	bAutomat4 := fbButtAuto4.bOutB  AND NOT bStartAutomat4 AND NOT bSound4;
	fbPuls(tPeriod := T#0.5S);

	fbButtManu4(bButt := bButtManu4 AND NOT  bAutomat4, bReset := bReset4 OR bAlarm4);
	bManual4 := fbButtManu4.bOutB;

	fbButtReverse4(bButt := bButtReverse4 AND NOT b_4KM1_1, bReset := bReset4 OR bAlarm4);
	bReverse4 := fbButtReverse4.bOutB;

	fbButtStop4(bButt := bButtStop4 OR bAlarm4, bReset := bReset4);
	bStop4 := fbButtStop4.bOutB ;
    	
	fbTimerStart4 (IN := bStartAutomat4, PT := T#1S);

IF NOT bStop4 AND fbTimerStart4.Q AND NOT 
  ( bDrive4s01M1 OR bDrive4s02M1 OR bDrive4s03M1 OR 
	bDrive4s04M1 OR bDrive4s05M1 OR bDrive4s06M1 OR 
	bDrive4s01M1Rev OR bDrive4s02M1Rev OR bDrive4s03M1Rev OR 
	bDrive4s04M1Rev OR bDrive4s05M1Rev OR bDrive4s06M1Rev )
THEN bStartAutomat4 := FALSE;
END_IF

IF bReset4 THEN bAutomat4 := FALSE; bManual4 := FALSE; bStop4 := FALSE; bStartAutomat4 := FALSE;
END_IF

fbpulse4(ENABLE := bStartAutomat4 OR bSound4,TIMELOW := T#500MS, TIMEHIGH:=T#500MS);
//Светофоры первого конвейера
bGreen_4S1HL1  := bAutomat4 AND NOT bManual4 AND NOT bAlarm4 AND NOT bSound4 OR fbpulse4.OUT;
bGreen_4S1_HL1 := bAutomat4 AND NOT bManual4 AND NOT bAlarm4 AND NOT bSound4 OR fbpulse4.OUT;

bYellow_4S1HL1 := NOT bAutomat4 AND bManual4 AND NOT bAlarm4;
bYellow_4S1_HL1:= NOT bAutomat4 AND bManual4 AND NOT bAlarm4;
//---------------------------------------------------------------------------------------------------//

ACTION ACT_Conversion:
Massa_1_INT :=REAL_TO_INT( Massa_1);
Massa_2_INT :=REAL_TO_INT( Massa_2);
Massa_3_INT :=REAL_TO_INT( Massa_3);
Massa_4_INT :=REAL_TO_INT( Massa_4);

Massa_1_Gramms := REAL_TO_DINT( Massa_1 * 1000000);
Massa_2_Gramms := REAL_TO_DINT( Massa_2 * 1000000);
Massa_3_Gramms := REAL_TO_DINT( Massa_3 * 1000000);
Massa_4_Gramms := REAL_TO_DINT( Massa_4 * 1000000);
END_ACTION

ACTION ACT_Drive:
//----------------------------------------------------------// конвейер 1
b1K2 := bDrive1s01M1 OR bDrive1s01M1Rev; // Пуск 1UZ1					 
b1K3 := bDrive1s02M1 OR bDrive1s02M1Rev; // Пуск 1UZ2
b1K4 := bDrive1s03M1 OR bDrive1s03M1Rev; // Пуск 1UZ3
b1K5 := bDrive1s04M1 OR bDrive1s04M1Rev; // Пуск 1UZ4
b1K6 := bDrive1s05M1 OR bDrive1s05M1Rev; // Пуск 1UZ5
b1K7 := bDrive1s06M1 OR bDrive1s06M1Rev; // Пуск 1UZ6
//---------------------------------------------------------// конвейер 2
b2K2 := bDrive2s01M1 OR bDrive2s01M1Rev; // Пуск 2UZ1					 
b2K3 := bDrive2s02M1 OR bDrive2s02M1Rev; // Пуск 2UZ2
b2K4 := bDrive2s03M1 OR bDrive2s03M1Rev; // Пуск 2UZ3
b2K5 := bDrive2s04M1 OR bDrive2s04M1Rev; // Пуск 2UZ4
b2K6 := bDrive2s05M1 OR bDrive2s05M1Rev; // Пуск 2UZ5
b2K7 := bDrive2s06M1 OR bDrive2s06M1Rev; // Пуск 2UZ6
//---------------------------------------------------------// конвейер 3
b3K2 := bDrive3s01M1 OR bDrive3s01M1Rev; // Пуск 3UZ1					 
b3K3 := bDrive3s02M1 OR bDrive3s02M1Rev; // Пуск 3UZ2
b3K4 := bDrive3s03M1 OR bDrive3s03M1Rev; // Пуск 3UZ3
b3K5 := bDrive3s04M1 OR bDrive3s04M1Rev; // Пуск 3UZ4
b3K6 := bDrive3s05M1 OR bDrive3s05M1Rev; // Пуск 3UZ5
b3K7 := bDrive3s06M1 OR bDrive3s06M1Rev; // Пуск 3UZ6
//---------------------------------------------------------// конвейер 4
b4K2 := bDrive4s01M1 OR bDrive4s01M1Rev; // Пуск 4UZ1					 
b4K3 := bDrive4s02M1 OR bDrive4s02M1Rev; // Пуск 4UZ2
b4K4 := bDrive4s03M1 OR bDrive4s03M1Rev; // Пуск 4UZ3
b4K5 := bDrive4s04M1 OR bDrive4s04M1Rev; // Пуск 4UZ4
b4K6 := bDrive4s05M1 OR bDrive4s05M1Rev; // Пуск 4UZ5
b4K7 := bDrive4s06M1 OR bDrive4s06M1Rev; // Пуск 4UZ6
END_ACTION

ACTION ACT_Light:
bSound_1S1HL1 := bSound1;
bSound_1S1_HL1:= bSound1;
bSound_2S1HL1 := bSound2;
bSound_2S1_HL1:= bSound2;
bSound_3S1HL1 := bSound3;
bSound_3S1_HL1:= bSound3;
bSound_4S1HL1 :=bSound4;
bSound_4S1_HL1:=bSound4;
END_ACTION

END_PROGRAM

// ---- POUs/FB/Puls.TcPOU
FUNCTION_BLOCK Puls

VAR_INPUT
 	EN 		:BOOL := TRUE;
    Period	:TIME;
END_VAR
VAR_OUTPUT
	Puls	:BOOL;
END_VAR
VAR
	M		:BOOL:=0;
	R1		:R_TRIG;
	t		:BOOL;
	R2		:R_TRIG;
	TP1		:TP;
	TP2		:TP;
	M1		:BOOL:=0;
END_VAR

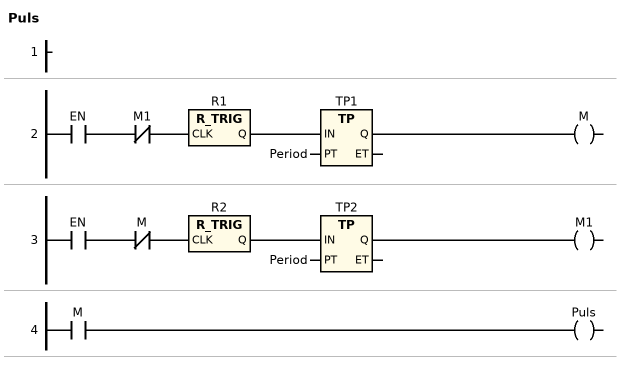
// NETWORK 1

// NETWORK 2
R1(CLK := EN AND NOT M1); // R_TRIG
TP1(IN := R1.Q, PT := Period); // TP
M := TP1.Q;

// NETWORK 3
R2(CLK := EN AND NOT M); // R_TRIG
TP2(IN := R2.Q, PT := Period); // TP
M1 := TP2.Q;

// NETWORK 4
Puls := M;

END_FUNCTION_BLOCK

// ---- POUs/FB/FBauxiliary/FB_ButtonToggle.TcPOU
FUNCTION_BLOCK FB_ButtonToggle
VAR_INPUT
	bReset  :BOOL;
	bEnable :BOOL := TRUE;
	bButt   :BOOL;
END_VAR
VAR
	fbButt  :R_TRIG;
END_VAR
VAR_OUTPUT
	bOutB   :BOOL;
END_VAR

fbButt(CLK:=bButt);

IF fbButt.Q AND bEnable THEN
	IF bOutB THEN bOutB := FALSE;
		ELSE bOutB := TRUE;
	END_IF
END_IF

IF bReset THEN bOutB := FALSE;
END_IF

END_FUNCTION_BLOCK

// ---- POUs/FB/FB_Puls.TcPOU
FUNCTION_BLOCK FB_Puls
VAR_INPUT
	tPeriod  :TIME;
END_VAR
VAR_OUTPUT
	bPuls 	 :BOOL;
END_VAR
VAR
	bM1		 :BOOL := TRUE;
	TP1		 :TP;
	TP2		 :TP;
	fbPulsM1 :F_TRIG;
	iCounter :INT;
	bM2		 :BOOL;
	fbPulsM2 :F_TRIG;
END_VAR

fbPulsM1(CLK:= bM1);
TP1(IN:= fbPulsM1.Q, PT:=tPeriod);
bM2 :=TP1.Q;

fbPulsM2(CLK:= bM2);
TP2(IN:= fbPulsM1.Q,  PT:=tPeriod);

bM1:= TP2.Q;
bPuls := bM1;
IF fbPulsM1.Q THEN
	iCounter:=iCounter+1;
END_IF

END_FUNCTION_BLOCK

// ---- POUs/TCP_IP.TcPOU
PROGRAM TCP_IP
VAR		 
	sSrvNetID	:T_AmsNetID := '';						/// TwinCAT TCP/IP server network address
	sLocalHost	:T_IPv4Addr := '10.45.19.80';			/// Own (server) IP address! 
	 
	nLocalPort1	:UDINT := 2001;							/// Own (server 1) port number!	
	nLocalPort2	:UDINT := 2002;							/// Own (server 2) port number!  
	nLocalPort3	:UDINT := 2003;							/// Own (server 3) port number!	 
	nLocalPort4	:UDINT := 2004;							/// Own (server 4) port number!
	 
	bEnable1	:BOOL  := TRUE;							/// TRUE => enable server 1(connection) instance, FALSE => disable
	bEnable2	:BOOL  := TRUE;							/// TRUE => enable server 2(connection) instance, FALSE => disable
	bEnable3	:BOOL  := TRUE;							/// TRUE => enable server 3(connection) instance, FALSE => disable
	bEnable4	:BOOL  := TRUE;							/// TRUE => enable server 4(connection) instance, FALSE => disable
	bEnable5	:BOOL  := TRUE;							/// TRUE => enable server  (connection) instance, FALSE => disable
	
	bLog		:BOOL  := TRUE;							/// TRUE => Enable error/message log, FALSE => Disable 
	 
	fbServer1	:FB_Server := (sPrefix := 'SERVER1::');	/// Application (connection) instance 1
	fbServer2	:FB_Server := (sPrefix := 'SERVER2::');	/// Application (connection) instance 2
	fbServer3	:FB_Server := (sPrefix := 'SERVER3::');	/// Application (connection) instance 3
	fbServer4	:FB_Server := (sPrefix := 'SERVER4::');	/// Application (connection) instance 4
	 
	hServer1	:T_HSERVER;								/// Server connection handle 1	
	hServer2	:T_HSERVER;								/// Server connection handle 2	
	hServer3	:T_HSERVER;								/// Server connection handle 3
	hServer4	:T_HSERVER; 							/// Server connection handle 4

	fbCloseAll	:FB_SocketCloseAll;
	bInitialize	:BOOL := TRUE;

END_VAR

IF bInitialize THEN
	bInitialize := FALSE;

	(* Initialize server handle once *)
	F_CreateServerHnd( 	sSrvNetID 	:= sSrvNetID, 
						sLocalHost 	:= sLocalHost, 
						nLocalPort	:= nLocalPort1,
						nMode 		:= SEL( bLog, 0, CONNECT_MODE_ENABLEDBG),	(* Enable/disable debug messages? *)
						bEnable 	:= FALSE,									(* TRUE = leave listener socket open, FALSE = close listener socket after last connection ist closed too *)
						hServer 	:= hServer1 );
						
	F_CreateServerHnd( 	sSrvNetID 	:= sSrvNetID, 
						sLocalHost 	:= sLocalHost, 
						nLocalPort	:= nLocalPort2,
						nMode 		:= SEL( bLog, 0, CONNECT_MODE_ENABLEDBG),	(* Enable/disable debug messages? *)
						bEnable 	:= FALSE,									(* TRUE = leave listener socket open, FALSE = close listener socket after last connection ist closed too *)
						hServer 	:= hServer2 );					
						
	F_CreateServerHnd( 	sSrvNetID 	:= sSrvNetID, 
						sLocalHost 	:= sLocalHost, 
						nLocalPort	:= nLocalPort3,
						nMode 		:= SEL( bLog, 0, CONNECT_MODE_ENABLEDBG),	(* Enable/disable debug messages? *)
						bEnable 	:= FALSE,									(* TRUE = leave listener socket open, FALSE = close listener socket after last connection ist closed too *)
						hServer 	:= hServer3 );					
						
	F_CreateServerHnd( 	sSrvNetID 	:= sSrvNetID, 
						sLocalHost 	:= sLocalHost, 
						nLocalPort	:= nLocalPort4,
						nMode 		:= SEL( bLog, 0, CONNECT_MODE_ENABLEDBG),	(* Enable/disable debug messages? *)
						bEnable 	:= FALSE,									(* TRUE = leave listener socket open, FALSE = close listener socket after last connection ist closed too *)
						hServer 	:= hServer4 );										
END_IF

fbServer1( hServer := hServer1, sSrvNetID := sSrvNetID, bEnable := bEnable1, bLog := bLog, 
  	bReadScan:=bReadScan_1,sScanID:=sScanID_1 );
fbServer2( hServer := hServer2, sSrvNetID := sSrvNetID, bEnable := bEnable2, bLog := bLog, 
  	bReadScan:=bReadScan_2,sScanID:=sScanID_2 );
fbServer3( hServer := hServer3, sSrvNetID := sSrvNetID, bEnable := bEnable3, bLog := bLog, 
	bReadScan:=bReadScan_3,sScanID:=sScanID_3 );
fbServer4( hServer := hServer4, sSrvNetID := sSrvNetID, bEnable := bEnable4, bLog := bLog, 
	bReadScan:=bReadScan_4,sScanID:=sScanID_4 );

b_1S4_2A2 := bRequestID_1;
b_2S4_2A2 := bRequestID_2;
b_3S4_2A2 := bRequestID_3;
b_4S4_2A2 := bRequestID_4;

END_PROGRAM

// ---- POUs/Ethernet/FB_Server.TcPOU
FUNCTION_BLOCK FB_Server
VAR_IN_OUT
	/// Server connection handle 
	hServer: T_HSERVER;
	bReadScan: BOOL;
	sScanID:STRING;
END_VAR
VAR_INPUT
	/// TwinCAT TCP/IP server network address 
	sSrvNetID: T_AmsNetID := '';
	/// TRUE => enable server data exchange, FALSE => disable 
	bEnable: BOOL := FALSE;
	/// TRUE => Enable log message output, FALSE => Disable 
	bLog: BOOL := TRUE;
	/// Log message description string (allows the identification of log message source) 
	sPrefix: STRING := 'SERVER::';
END_VAR
VAR_OUTPUT
	/// TCP/IP connection state 
	eState: E_SocketConnectionState := eSOCKET_DISCONNECTED;
	
END_VAR
VAR
	/// Server application control function block 
	fbApplication: FB_ServerApplication;
	/// Server data exchange control function block. Implements one server<->client connection 
	fbConnection: FB_ServerConnection;
	/// Tx fifo 
	fbTx: FB_FrameFifo;
	/// Rx fifo 
	fbRx: FB_FrameFifo;
	/// Log/debug/error fifo 
	fbLog: FB_LogFifo;
END_VAR

(*-------------------------------- Trigger data exchange -----------------------------------------*)
fbConnection( hServer := hServer, sSrvNetID := sSrvNetID, fbRx := fbRx, fbTx := fbTx, fbLog := fbLog, 
			bEnable := bEnable, bLog := bLog, sPrefix := sPrefix, eState => eState );
IF fbConnection.eState = eSOCKET_CONNECTED THEN(* Connection established *)
	fbApplication( fbTx := fbTx, fbRx := fbRx, fbLog := fbLog,bReadScan:=bReadScan,sFromClient:= sScanID  );
	
END_IF

END_FUNCTION_BLOCK

// ---- POUs/Ethernet/FB_ServerApplication.TcPOU
///----------------------- Simple TCP/IP application. Adapt this code to match your needs. ----
FUNCTION_BLOCK FB_ServerApplication
VAR_IN_OUT
	/// TX fifo 
	fbTx: FB_FrameFifo;
	/// RX fifo 
	fbRx: FB_FrameFifo;
	/// Log/debug/error fifo 
	fbLog: FB_LogFifo;
	bReadScan: BOOL;
	sFromClient: STRING;
END_VAR
VAR
	sToClient: T_MaxString := '';
	sLogMessage: T_MaxString := '';
	nCounter: UDINT;
	sFrom_Client:STRING;
END_VAR
VAR_OUTPUT
	
END_VAR

(*------------------------------- Get received message strings ------------------------------------------*)
REPEAT

	fbRx.RemoveHead( );(* Fetch received string from rx fifo *)
	IF fbRx.bOk THEN(* Success *)

		(*TODO: Implement receive data handler *)
	//	nCounter := nCounter + 1;
		sFrom_Client := fbRx.sGet;
		sFromClient:= LEFT(sFrom_Client,LEN(sFrom_Client)-2 );
		bReadScan:=TRUE;
	//	sToClient 	:= sFromClient;

		(* Send received string back to the client *)
	(*	fbTx.AddTail( sPut := sToClient );(* Add string to the tx fifo *)
		IF NOT fbTx.bOk THEN(* Fifo overflow => log error *)
			fbLog.Error( sMessage := 'FB_FrameFifo(sender)', nErrID := PLCPRJ_ERROR_SENDFIFO_OVERFLOW );
		END_IF*)
	END_IF

UNTIL NOT fbRx.bOk
END_REPEAT



(*------------------------------- Get log/error messages from log fifo ----------------------------------------*)
REPEAT
	fbLog.Remove( );
	IF fbLog.bOk THEN

		(* TODO: Implement log message handler *)
		sLogMessage := fbLog.sGet;

	END_IF
UNTIL NOT fbLog.bOk
END_REPEAT

END_FUNCTION_BLOCK

// ---- POUs/Ethernet/Helper POUs/FB_FrameFifo.TcPOU
(* Tx/Rx (string data) fifo control function block *)
FUNCTION_BLOCK FB_FrameFifo
VAR_INPUT
	bLog		: BOOL			:= FALSE; (* TRUE => Enable debug output, FALSE => Disable *)
	sPrefix		: STRING		:= 'Unknown::';(* Debug message description string (allows the identification of log message source) *)
	sPut		: T_MaxString 	:= ''; (* String to add (write) to the buffer *)
END_VAR
VAR_OUTPUT
	bOk			: BOOL; 	 	(* TRUE = New entry added or removed succesfully, FALSE = Fifo overflow or fifo empty *)
	sGet		: T_MaxString 	:= '';(* String removed (read) from buffer *)
	nCount		: UDINT			:= 0;(* Number of fifo entries *)
	cbFree		: UDINT 		:= 0;(* Free buffer space *)
END_VAR
VAR
	fbBuffer 	: FB_StringRingBuffer := (bOverwrite := FALSE);(* Basic (lower level) string buffer control function block *)
	buffer		: ARRAY[-3..PLCPRJ_BUFFER_SIZE] OF BYTE;(* Internal buffer memory *)
END_VAR

;

ACTION AddTail:
(* Adds new fifo entry *)
fbBuffer.A_AddTail( pBuffer:= ADR(buffer), cbBuffer:= SIZEOF(buffer),
					putValue:= sPut, bOk=>bOk, nCount=>nCount );
IF bOk THEN
	cbFree := PLCPRJ_BUFFER_SIZE - fbBuffer.cbSize;(* Calculate the free buffer space *)
	IF bLog THEN(* Log message *)
		ADSLOGSTR( ADSLOG_MSGTYPE_HINT OR ADSLOG_MSGTYPE_LOG, CONCAT( sPrefix, '<="%s"' ), sPut );
	END_IF
END_IF
END_ACTION

ACTION Clear:
(* Resets fifo = clears all data *)
fbBuffer.A_Reset( pBuffer:= ADR(buffer), cbBuffer:= SIZEOF(buffer),
				bOk=>bOk, getValue=>sGet, nCount=>nCount );
cbFree := PLCPRJ_BUFFER_SIZE;(* Free buffer size *)
END_ACTION

ACTION RemoveHead:
(* Removes oldest fifo entry *)
fbBuffer.A_RemoveHead( pBuffer:= ADR(buffer), cbBuffer:= SIZEOF(buffer),
						bOk=>bOk, getValue=>sGet, nCount=>nCount );
IF bOk THEN
	cbFree := PLCPRJ_BUFFER_SIZE - fbBuffer.cbSize;(* Calculate the free buffer space *)
END_IF
END_ACTION

END_FUNCTION_BLOCK

// ---- POUs/Ethernet/Helper POUs/FB_LogFifo.TcPOU
(* Log/debug/error message fifo *)
FUNCTION_BLOCK FB_LogFifo
VAR_INPUT
	bLog		: BOOL 		:= FALSE;(* TRUE => Enable log message output, FALSE => Disable *)
	sPrefix		: STRING 	:= 'Unknown::';(* Log message description string (allows the identification of log message source) *)
	
	sMessage	: STRING 	:= '';(* String message to add (write) to the fifo *)
	nErrID		: UDINT 	:= 0;(* Error code to add (write) to the fifo *)
	hSocket		: T_HSOCKET;(* Socket connection handle *)
END_VAR
VAR_OUTPUT
	bOk			: BOOL;(* TRUE = New entry added or removed succesfully, FALSE = Fifo overflow or fifo empty *)
	sGet		: T_MaxString := '';(* String entry removed (read) from fifo *)
	nCount		: UDINT := 0;(* Number of fifo entries *)
END_VAR
VAR
	fbBuffer 	: FB_StringRingBuffer;(* Basic (lower level) string buffer control function block *)
	buffer		: ARRAY[0..PLCPRJ_BUFFER_SIZE] OF BYTE;(* Internal buffer memory *)
	sSource		: T_MaxString;	
	sPut		: T_MaxString;
END_VAR

;

ACTION Clear:
(* Clears all fifo entries *)
fbBuffer.A_Reset( 	pBuffer := ADR( buffer ), cbBuffer := SIZEOF( buffer ), 
					bOk=>bOk, nCount=>nCount, getValue=>sGet );
END_ACTION

ACTION Error:
(* Adds new fifo entry *)
IF nErrID = 0 THEN
	sSource := '::Error: 0x';
ELSIF ( nErrID AND 16#80000000) = 16#80000000 THEN
	IF nErrID = 16#80072746 THEN
		sSource := '::Win32 error (the connection is reset by remote side): 0x';
	ELSE
		sSource := '::Win32 error: 0x';
	END_IF
ELSIF (nErrID AND 16#00008100) = 16#00008100 THEN
	CASE nErrID OF
		PLCPRJ_ERROR_RECEIVE_TIMEOUT:
			sSource := '::PLC sample project receive timeout error: 0x';
		PLCPRJ_ERROR_SENDFIFO_OVERFLOW:
			sSource := '::PLC sample project send fifo overflow error: 0x';
		PLCPRJ_ERROR_RECFIFO_OVERFLOW:
			sSource := '::PLC sample project receive fifo overflow error: 0x';
	ELSE
		sSource := '::Other PLC sample project error: 0x';
	END_CASE
ELSIF (nErrID AND 16#00008000) = 16#00008000 THEN
	sSource := '::Internal TCP/IP Connection Server error: 0x';
ELSE
	sSource := '::TwinCAT System error: 0x';
END_IF

sPut := CONCAT( CONCAT( CONCAT( sPrefix, sMessage ), sSource ), DWORD_TO_HEXSTR( nErrID AND 16#FFFF, 0, FALSE ) ); 

fbBuffer.A_AddTail( pBuffer:= ADR(buffer), cbBuffer:= SIZEOF(buffer),
					putValue:= sPut, bOk=>bOk, nCount=>nCount );
IF bOk THEN
	IF bLog THEN(* Log error message *)
		ADSLOGSTR( ADSLOG_MSGTYPE_ERROR OR ADSLOG_MSGTYPE_LOG, '%s', sPut );	
	END_IF
END_IF
END_ACTION

ACTION Message:
(* Adds new fifo entry *)
sPut := CONCAT( CONCAT( sPrefix, sMessage ), CONCAT( '::', HSOCKET_TO_STRING(hSocket) ) );
fbBuffer.A_AddTail( pBuffer:= ADR(buffer), cbBuffer:= SIZEOF(buffer),
					putValue:= sPut, bOk=>bOk, nCount=>nCount );
IF bOk THEN
	IF bLog THEN(* Log information message *)
		ADSLOGSTR( ADSLOG_MSGTYPE_HINT OR ADSLOG_MSGTYPE_LOG, '%s', sPut );	
	END_IF
END_IF
END_ACTION

ACTION Remove:
(* Removes oldest fifo entry *)
IF nCount = 0 THEN
	sGet := '';
	bOk := FALSE;
	RETURN;
END_IF

fbBuffer.A_RemoveHead( pBuffer:= ADR(buffer), cbBuffer:= SIZEOF(buffer),
						getValue=>sGet, bOk=>bOk, nCount=>nCount );
END_ACTION

END_FUNCTION_BLOCK

// ---- POUs/Ethernet/FB_ServerConnection.TcPOU
/// This function block implements simple TCP/IP server protocol. 
FUNCTION_BLOCK FB_ServerConnection
VAR_IN_OUT
	/// Server connection handle 
	hServer: T_HSERVER;
	/// TX fifo 
	fbTx: FB_FrameFifo;
	/// RX fifo 
	fbRx: FB_FrameFifo;
	/// Log/debug/error fifo 
	fbLog: FB_LogFifo;
END_VAR
VAR_INPUT
	/// TwinCAT TCP/IP server network address 
	sSrvNetID: T_AmsNetID := '';
	/// TRUE => Enable/connect, FALSE => Disable/disconnect 
	bEnable: BOOL := FALSE;
	/// Try to reconnect after this time 
	tReconnect: TIME := TIME#1s0ms;
	/// TRUE => Enable log message output, FALSE => Disable 
	bLog: BOOL := FALSE;
	/// Log message description string (allows the identification of log message source) 
	sPrefix: STRING := 'SERVER::';
END_VAR
VAR_OUTPUT
	/// TCP/IP connection state 
	eState: E_SocketConnectionState := eSOCKET_DISCONNECTED;
END_VAR
VAR
	/// Create/release TCP/IP connection 
	fbConnect: FB_ServerClientConnection;
	/// Send TCP/IP data 
	fbSend: FB_SocketSend;
	/// Receive TCP/IP data 
	fbReceive: FB_SocketReceive;
	/// Global state 
	nState: BYTE;
	/// Tx state 
	bSndBusy: BOOL;
	/// Rx state 
	bRcvBusy: BOOL;
	/// Disconnect flag, if set the socket will be closed 
	bDisconnect: BOOL;
	/// Receive poll timer 
	fbPollTimer: TON;
	/// Request timeout timer 
	fbRequestTimer: TON;
	/// Reconnect timer 
	fbReconnectTimer: TON;
	/// Count of received data bytes 
	cbReceived: UDINT;
	/// Byte length of received string 
	cbRx: UDINT;
	/// Temp. RX buffer 
	buffer: ARRAY[0..PLCPRJ_BUFFER_SIZE] OF BYTE;
	sTxFrame: T_MaxString;
	sRxFrame: T_MaxString;
	i: UDINT;
	bAbort: BOOL;
	bTest:BOOL;
END_VAR

CASE nState OF
	0:(* Connect *)
		fbConnect( 	eMode := eACCEPT_ALL, tReconnect := tReconnect, bEnable := bEnable, 
					hServer := hServer, eState => eState );
		IF NOT fbConnect.bBusy THEN
			IF NOT fbConnect.bError THEN
				IF eState = eSOCKET_CONNECTED THEN(* We are connected *)

					fbTx.Clear( sPrefix := CONCAT( sPrefix, 'FB_FrameFifo(sender)::' ), bLog := bLog );(* Clear TX fifo (optional) *)
					fbRx.Clear( sPrefix := CONCAT( sPrefix, 'FB_FrameFifo(receiver)::' ), bLog := bLog );(* Clear RX fifo (optional) *)
					fbLog.Clear( sPrefix := sPrefix, bLog := bLog );(* Clear log fifo (optional) *)
					bSndBusy := FALSE;
					bRcvBusy := FALSE;
					bDisconnect := FALSE;
					cbReceived := 0;

					fbPollTimer( IN := FALSE, PT := T#0S );
					fbRequestTimer( IN := FALSE, PT := PLCPRJ_RECEIVE_TIMEOUT );
					fbReconnectTimer( IN := FALSE, PT := tReconnect );

					fbLog.Message( sMessage := 'Connection established!', hSocket := fbConnect.hSocket );
					nState := 1;
				END_IF
			ELSE(* Error => log error *)
				fbLog.Error( sMessage := 'FB_ServerClientConnection()', nErrID := fbConnect.nErrID );
			END_IF
		END_IF

	1:(* Data exchange state *)
	bTest:=TRUE;
		bDisconnect := NOT bEnable OR bDisconnect;(* User/internal disconnect requested? *)
		IF bDisconnect AND NOT bSndBusy AND NOT bRcvBusy THEN
			bDisconnect := FALSE;
			fbLog.Message( sMessage := 'Closing connection!', hSocket := fbConnect.hSocket );
			nState := 2;(* Disconnect *)
		ELSE

			(* ------------------------ Get rx data --------------------------------------- *)
			IF NOT bDisconnect AND NOT bRcvBusy THEN

				fbPollTimer( IN := TRUE );
				IF fbPollTimer.Q THEN
					IF fbRx.cbFree >= SIZEOF(sRxFrame) THEN(* Check free rx fifo space *)
						fbPollTimer( IN := FALSE, PT := PLCPRJ_RECEIVE_POLLING_TIME );
						fbReceive( bExecute := FALSE );
						fbReceive( sSrvNetId	:= sSrvNetID,
									hSocket		:= fbConnect.hSocket,
									cbLen		:= SIZEOF(buffer) - cbReceived,
									pDest		:= ADR(buffer) + cbReceived,
									bExecute	:= TRUE );
						bRcvBusy := TRUE;
					END_IF
				END_IF
				
			ELSE(* Wait until receive not busy *)
				
				fbReceive( bExecute := FALSE );
				IF NOT fbReceive.bBusy THEN
					bRcvBusy := FALSE;
					IF NOT fbReceive.bError THEN
						IF fbReceive.nRecBytes > 0 THEN(* Bytes received *)
							
							fbPollTimer( IN := FALSE, PT := T#0S );(* Bytes received => increase the read (polling) speed *)
							fbRequestTimer( IN := FALSE );(* Bytes received => disable timeout check *)
							cbReceived := cbReceived + fbReceive.nRecBytes;(* Calculate the number of received data bytes *)

							(* Parse received bytes and extract strings *)
							REPEAT
								bAbort := TRUE;(* Set flag *)
								IF cbReceived > 0 THEN

									(* Search for string null delimiter *)
									FOR i:= 0 TO cbReceived - 1 BY 1 DO
										IF buffer[i] = 0 THEN (* End of string position found *)

											cbRx := i + 1;(* Calculate the length of string (inclusive the end delimiter) *)
											MEMCPY( ADR(sRxFrame), ADR(buffer), MIN(cbRx, SIZEOF(sRxFrame) ) );(* Copy string bytes to fifo input variable *)

											fbRx.AddTail( sPut := sRxFrame );(* Add string to the rx fifo *)
											IF fbRx.bOk THEN

												MEMMOVE( ADR(buffer), ADR(buffer) + cbRx, cbReceived - cbRx );(* Move/shift remaining bytes in buffer *)
												cbReceived := cbReceived - cbRx;(* Recalculate the remaining data length *)

												IF fbRx.cbFree >= SIZEOF(sRxFrame) THEN(* Check free rx fifo space *)
													bAbort := FALSE;(* Reset flag, try to parse the next string  *)
												END_IF

											ELSE(* Fifo overflow => log error and disconnect *)
												fbLog.Error( sMessage := 'FB_FrameFifo(receiver)', nErrID := PLCPRJ_ERROR_RECFIFO_OVERFLOW );
												bDisconnect := TRUE;(* Set flag *)
												RETURN;
											END_IF

											EXIT;
										END_IF
									END_FOR

								END_IF (* IF cbReceived > 0 THEN *)

							UNTIL bAbort
							END_REPEAT

						ELSE(* No bytes received *)
							fbRequestTimer( IN := TRUE );(* No bytes received => enable timeout check *)
							IF fbRequestTimer.Q THEN (* Timeout error*)
								fbRequestTimer( IN := FALSE );
								fbLog.Error( sMessage := 'FB_SocketReceive()', nErrID := PLCPRJ_ERROR_RECEIVE_TIMEOUT );
								bDisconnect := TRUE;(* Set flag *)
							END_IF							
						END_IF(* IF fbReceive.nRecBytes > 0 THEN *)
					ELSE(* Receive error => log error and disconnect *)
						fbLog.Error( sMessage := 'FB_SocketReceive()', nErrID := fbReceive.nErrId );
						bDisconnect := TRUE;(* Set flag *)
					END_IF
				END_IF
			
			END_IF(* IF NOT bDisconnect AND NOT bRcvBusy THEN *)
			(* ---------------------------------------------------------------------------- *)


			(* --------------------------- Send tx data ----------------------------------- *)
		(*	IF NOT bDisconnect AND NOT bSndBusy THEN
				fbTx.RemoveHead( sGet => sTxFrame );(* Remove oldest string entry s*)
				IF fbTx.bOk THEN(* Success *)
					fbSend( bExecute := FALSE );
					fbSend(	sSrvNetID 	:= sSrvNetID,
							hSocket		:= fbConnect.hSocket,
							cbLen		:= INT_TO_UDINT(LEN( sTxFrame )) + 1,(* Send string inclusive string (null) delimiter! *)
							pSrc		:= ADR( sTxFrame ),(* Address of the string variable *)
							bExecute	:= TRUE );
					bSndBusy := TRUE;
				END_IF
			ELSE(* Wait until send not busy *)
				fbSend( bExecute := FALSE );
				IF NOT fbSend.bBusy THEN
					bSndBusy := FALSE;
					IF fbSend.bError THEN(* Send error => log error and disconnect *)
						fbLog.Error( sMessage := 'FB_SocketSend()', nErrID := fbSend.nErrId );
						bDisconnect := TRUE;(* Set flag *)
					END_IF
				END_IF
			END_IF(* IF NOT bDisconnect AND NOT bSndBusy THEN *)
			*)
			(* ---------------------------------------------------------------------------- *)

			
		END_IF(* IF bDisconnect AND NOT bSndBusy AND NOT bRcvBusy THEN *)


	2:(* Disconnect *)
		fbConnect( hServer := hServer, bEnable:= FALSE, eState=>eState );
		IF eState = eSOCKET_DISCONNECTED THEN
			fbReconnectTimer( IN := TRUE );(* Please wait some seconds and then try to connect again *)
			IF fbReconnectTimer.Q THEN
				fbReconnectTimer( IN := FALSE );
				nState := 0;
			END_IF
		END_IF

END_CASE

END_FUNCTION_BLOCK

// ---- POUs/Alarms/Alarm_conv_1.TcPOU
PROGRAM Alarm_conv_1
VAR
timer1 : TON;
timer2 : TON;
timer3 : TON;
timer4 : TON;
timer5 : TON;
timer6 : TON;

bAlarm_b1_S1_SB0_blink	:BOOL;
bAlarm_b1_S6_SB0_blink	:BOOL;

Blinking				:BOOL :=TRUE;
END_VAR

//Нет готовности конвейер 1
	bAlarm1QF2_1QF7 S=NOT b_1QF2_1QF7 	AND bPermAlarm1;
	bAlarm1QF8 		S=NOT b_1QF8 		AND bPermAlarm1;
//	bAlarm1KM2 		S=NOT b_1KM2 		AND bPermAlarm1;
//	bAlarm1KM3 		S=NOT b_1KM3 		AND bPermAlarm1;
//	bAlarm1KM4 		S=NOT b_1KM4 		AND bPermAlarm1;
//	bAlarm1KM5 		S=NOT b_1KM5 		AND bPermAlarm1;
//	bAlarm1KM6 		S=NOT b_1KM6 		AND bPermAlarm1;
//	bAlarm1KM7 		S=NOT b_1KM7 		AND bPermAlarm1;

//Грибки	
	bAlarm_b1_S1_SB0 S=NOT   b1_S1_SB0 	AND bPermAlarm1;
	bAlarm_b1_S6_SB0 S=NOT   b1_S6_SB0 	AND bPermAlarm1;

// Индикация на грибках
	b1S1_SB0 := NOT b1_S1_SB0 AND blink.OUT;
	b1S6_SB0 := NOT b1_S6_SB0 AND blink.OUT;
		
	blink(ENABLE:=Blinking,TIMELOW:=T#500MS,TIMEHIGH:=T#500MS);
	bAlarm_b1_S1_SB0_blink := blink.OUT AND bAlarm_b1_S1_SB0;
	bAlarm_b1_S6_SB0_blink := blink.OUT AND bAlarm_b1_S6_SB0;

	
(*Авария безопасности*)
	bAlarmSafety1 := bAlarm_b1_S1_SB0 OR bAlarm_b1_S6_SB0;

(*Нет общей готовности конвейера 1*)
	bNotReady_1 := bAlarm1QF2_1QF7 OR bAlarm1QF8 OR bAlarm1KM2 OR bAlarm1KM3 OR bAlarm1KM4 OR bAlarm1KM5 OR bAlarm1KM6 OR bAlarm1KM7;
					

IF  bNotReady1 THEN  sAlarm1:="Нет готовности 1";
		ELSIF bAlarmSafety1 THEN  sAlarm1:="Авария безопасности 1";
			ELSE sAlarm1:="---------";
END_IF

	bPermAlarmDrive1 := bPermAlarm1 AND NOT bAlarmSafety1;
	
(*(*Готовность *)
	IF NOT bDriveReady1s01M1 AND bPermAlarmDrive1  THEN  bNotDriveReady1s01M1 := TRUE;
	END_IF    
	IF NOT bDriveReady1s02M1 AND bPermAlarmDrive1  THEN  bNotDriveReady1s02M1 := TRUE;
	END_IF 
	IF NOT bDriveReady1s03M1 AND bPermAlarmDrive1  THEN  bNotDriveReady1s03M1 := TRUE;
	END_IF 
	IF NOT bDriveReady1s04M1 AND bPermAlarmDrive1  THEN  bNotDriveReady1s04M1 := TRUE;
	END_IF 
	IF NOT bDriveReady1s05M1 AND bPermAlarmDrive1  THEN  bNotDriveReady1s05M1 := TRUE;
	END_IF 
	IF NOT bDriveReady1s06M1 AND bPermAlarmDrive1  THEN  bNotDriveReady1s06M1 := TRUE;
	END_IF *)
	
(*Долгие перемещения Drive*)
	IF bLongMove1s01_s02_1   THEN bLongMove_1s01_s02_1 := TRUE;
	END_IF
	IF bLongMove1s02_1_s02_2  THEN bLongMove_1s02_1_s02_2 := TRUE;
	END_IF
	IF bLongMove1s02_2_s03_1  THEN bLongMove_1s02_2_s03_1 := TRUE;
	END_IF
	IF bLongMove1s02_s03  THEN bLongMove_1s02_s03 := TRUE;
	END_IF
		IF bLongMove1s03_1_s03_2   THEN bLongMove_1s03_1_s03_2 := TRUE;
	END_IF
	IF bLongMove1s03_2_s04_1  THEN bLongMove_1s03_2_s04_1 := TRUE;
	END_IF
	IF bLongMove1s03_s04  THEN bLongMove_1s03_s04 := TRUE;
	END_IF
	IF bLongMove1s04_1_s04_2  THEN bLongMove_1s04_1_s04_2 := TRUE;
	END_IF
		IF bLongMove1s04_2_s05   THEN bLongMove_1s04_2_s05  := TRUE;
	END_IF
	IF bLongMove1s05_1s06  THEN bLongMove_1s05_1s06 := TRUE;	
	END_IF

(*Нет готовности*)
	bNotReady1 := bNotDriveReady1s01M1 OR bNotDriveReady1s02M1 OR bNotDriveReady1s03M1 OR
			  bNotDriveReady1s04M1 OR bNotDriveReady1s05M1 OR bNotDriveReady1s06M1;

(*Долгое премещение*)
	bLongMove1 := bLongMove_1s02_1_s02_2 OR bLongMove_1s02_1_s02_2  OR bLongMove_1s02_s03 OR
	       bLongMove_1s03_1_s03_2 OR bLongMove_1s03_2_s04_1 OR bLongMove_1s03_s04 OR bLongMove_1s04_1_s04_2 OR
			bLongMove_1s04_2_s05   OR bLongMove_1s05_1s06;

(*Сброс бита аварии по кнопке с панели*)
	bAlarmReset1 := bButtAlarmReset1;
	
(*Восстановление/сброс аварийных сигналов*)
IF bReset1 OR bAlarmReset1 THEN
	bAlarm1QF8 :=FALSE; bAlarm1QF2_1QF7 :=FALSE;
	bAlarm1KM2 :=FALSE; bAlarm1KM3 :=FALSE; bAlarm1KM4 :=FALSE; bAlarm1KM5 :=FALSE; bAlarm1KM6 :=FALSE; bAlarm1KM7 :=FALSE;

	bNotDriveReady1s01M1 := FALSE; bNotDriveReady1s02M1 := FALSE; bNotDriveReady1s03M1 := FALSE;
	bNotDriveReady1s04M1 := FALSE; bNotDriveReady1s05M1 := FALSE; bNotDriveReady1s06M1 := FALSE;
	
	bLongMove_1s02_1_s02_2 := FALSE;bLongMove_1s02_1_s02_2 := FALSE; bLongMove_1s02_s03 := FALSE;
	bLongMove_1s03_1_s03_2 := FALSE; bLongMove_1s03_2_s04_1:= FALSE; bLongMove_1s03_s04 := FALSE;
	 bLongMove_1s04_1_s04_2:= FALSE;  bLongMove_1s04_2_s05 := FALSE;
    bLongMove_1s05_1s06 := FALSE;
	

	b1K2_b1KM2_err := FALSE; b1K3_b1KM3_err := FALSE; b1K4_b1KM4_err := FALSE;
	b1K5_b1KM5_err := FALSE; b1K6_b1KM6_err := FALSE; b1K7_b1KM7_err := FALSE;

	bAlarm_b1_S1_SB0	:= FALSE; bAlarm_b1_S6_SB0	:= FALSE;
END_IF

(*Формирование аварии*)
	bAlarm1 := bNotReady1 OR bLongMove1 OR bAlarmSafety1 OR bNotReady_1 OR bNotReadyGeneral OR bOverflow_CTU_Weight1 OR bOverflow_CTU_ID1;
	bAlarm1_vis := blink.OUT AND bAlarm1;

IF  bNotReady1 THEN  sAlarmLine1:="Нет готовности";
		ELSIF bLongMove1 THEN   sAlarmLine1:="Долгое перемещение";
			ELSE sAlarmLine1:="---------";
END_IF

IF bAlarm1 OR bStop1 THEN bRed_1S1HL1 :=TRUE; bRed_1S1_HL1 := TRUE;
	ELSE bRed_1S1HL1 := FALSE; bRed_1S1_HL1 := FALSE;
END_IF

AlarmEvent_conv1();
ACT1();

ACTION ACT1:
(*Контроль расцепления тормозов при включении двигателей*)	

//Контроль на секции 1
timer1(IN:=b1K2_b1KM2_bad,PT:=T#1000MS);

b1K2_b1KM2_good := b1K2 AND b_1KM2;
b1K2_b1KM2_bad := b1K2 AND NOT b_1KM2;

IF b1K2_b1KM2_bad AND timer1.Q THEN b1K2_b1KM2_err := TRUE;
END_IF
//-------------------------------------------------------//
//Контроль на секции 2
timer2(IN:=b1K3_b1KM3_bad,PT:=T#1000MS);

b1K3_b1KM3_good := b1K3 AND b_1KM3;
b1K3_b1KM3_bad := b1K3 AND NOT b_1KM3;

IF b1K3_b1KM3_bad AND timer2.Q THEN b1K3_b1KM3_err := TRUE;
END_IF
//-------------------------------------------------------//
//Контроль на секции 3
timer3(IN:=b1K4_b1KM4_bad,PT:=T#1000MS);

b1K4_b1KM4_good := b1K4 AND b_1KM4;
b1K4_b1KM4_bad := b1K4 AND NOT b_1KM4;

IF b1K4_b1KM4_bad AND timer3.Q THEN b1K4_b1KM4_err := TRUE;
END_IF
//-------------------------------------------------------//
//Контроль на секции 4
timer4(IN:=b1K5_b1KM5_bad,PT:=T#1000MS);

b1K5_b1KM5_good := b1K5 AND b_1KM5;
b1K5_b1KM5_bad := b1K5 AND NOT b_1KM5;

IF b1K5_b1KM5_bad AND timer4.Q THEN b1K5_b1KM5_err := TRUE;
END_IF
//-------------------------------------------------------//
//Контроль на секции 5
timer5(IN:=b1K6_b1KM6_bad,PT:=T#1000MS);

b1K6_b1KM6_good := b1K6 AND b_1KM6;
b1K6_b1KM6_bad := b1K6 AND NOT b_1KM6;

IF b1K6_b1KM6_bad AND timer5.Q THEN b1K6_b1KM6_err := TRUE;
END_IF
//-------------------------------------------------------//
//Контроль на секции 6
timer6(IN:=b1K7_b1KM7_bad,PT:=T#1000MS);

b1K7_b1KM7_good := b1K7 AND b_1KM7;
b1K7_b1KM7_bad := b1K7 AND NOT b_1KM7;

IF b1K7_b1KM7_bad AND timer6.Q THEN b1K7_b1KM7_err := TRUE;
END_IF
END_ACTION

END_PROGRAM

// ---- POUs/Alarms/AlarmEvent_conv1.TcPOU
PROGRAM AlarmEvent_conv1
VAR
	bIsInitalized				:BOOL;
	fbButtAlarmReset1_RTRIG 	:R_TRIG;

//готовность конвейера
	fbAlarm1QF2_1QF7			:FB_TcAlarm;
	fbAlarm1QF8					:FB_TcAlarm;
	fbAlarm1KM2					:FB_TcAlarm;
	fbAlarm1KM3					:FB_TcAlarm;
	fbAlarm1KM4					:FB_TcAlarm;
	fbAlarm1KM5					:FB_TcAlarm;
	fbAlarm1KM6					:FB_TcAlarm;
	fbAlarm1KM7					:FB_TcAlarm;	
//Контроль работы тормозов
	fbAlarm_b1K2_b1KM2_err		:FB_TcAlarm;
	fbAlarm_b1K3_b1KM3_err		:FB_TcAlarm;
	fbAlarm_b1K4_b1KM4_err		:FB_TcAlarm;
	fbAlarm_b1K5_b1KM5_err		:FB_TcAlarm;
	fbAlarm_b1K6_b1KM6_err		:FB_TcAlarm;
	fbAlarm_b1K7_b1KM7_err		:FB_TcAlarm;
//Грибки	
	fbAlarm_b1_S1_SB0			:FB_TcAlarm;
	fbAlarm_b1_S6_SB0			:FB_TcAlarm;
//готовность двигателей
	fbNotDriveReady1s01M1		:FB_TcAlarm;
	fbNotDriveReady1s02M1		:FB_TcAlarm;
	fbNotDriveReady1s03M1		:FB_TcAlarm;
	fbNotDriveReady1s04M1		:FB_TcAlarm;
	fbNotDriveReady1s05M1		:FB_TcAlarm;
	fbNotDriveReady1s06M1		:FB_TcAlarm;
//Долгие перемещения

	
	fbLongMove_1s01_s02_1	:FB_TcAlarm;
	fbLongMove_1s01_s02	    :FB_TcAlarm;
	fbLongMove_1s02_1_s02_2	:FB_TcAlarm;
	fbLongMove_1s02_2_s03_1	:FB_TcAlarm;
	fbLongMove_1s02_s03  	:FB_TcAlarm;
	fbLongMove_1s03_1_s03_2	:FB_TcAlarm;	
	fbLongMove_1s03_2_s04_1	:FB_TcAlarm;	
	fbLongMove_1s03_s04	    :FB_TcAlarm;	
	fbLongMove_1s04_1_s04_2	:FB_TcAlarm;
	fbLongMove_1s04_2_s05	:FB_TcAlarm;
	fbLongMove_1s05_1s06	:FB_TcAlarm;
	
	
	
//----------------------------------------------------------------------------//	
//готовность конвейера
	fbExecAlarm1QF2_1QF7		:FB_AlarmEvent;
	fbExecAlarm1QF8				:FB_AlarmEvent;
	fbExecAlarm1KM2				:FB_AlarmEvent;
	fbExecAlarm1KM3				:FB_AlarmEvent;
	fbExecAlarm1KM4				:FB_AlarmEvent;
	fbExecAlarm1KM5				:FB_AlarmEvent;
	fbExecAlarm1KM6				:FB_AlarmEvent;
	fbExecAlarm1KM7				:FB_AlarmEvent;
//Грибки	
	fbExecAlarm_b1_S1_SB0		:FB_AlarmEvent;
	fbExecAlarm_b1_S6_SB0		:FB_AlarmEvent;
//готовность двигателей
	fbExecNotDriveReady1s01M1	:FB_AlarmEvent;
	fbExecNotDriveReady1s02M1	:FB_AlarmEvent;
	fbExecNotDriveReady1s03M1	:FB_AlarmEvent;
	fbExecNotDriveReady1s04M1	:FB_AlarmEvent;
	fbExecNotDriveReady1s05M1	:FB_AlarmEvent;
	fbExecNotDriveReady1s06M1	:FB_AlarmEvent;
//Долгие перемещения
	fbExecLongMove_1s01_s02_1	:FB_AlarmEvent;
	fbExecLongMove_1s01_s02	 :FB_AlarmEvent;
	fbExecbLongMove_1s02_1_s02_2	:FB_AlarmEvent;
	fbExecLongMove_1s02_2_s03_1	:FB_AlarmEvent;
	fbExecLongMove_1s02_s03  	:FB_AlarmEvent;
	fbExecLongMove_1s03_1_s03_2	:FB_AlarmEvent;	
	fbExecLongMove_1s03_2_s04_1	:FB_AlarmEvent;	
	fbExecLongMove_1s03_s04	:FB_AlarmEvent;	
	fbExecLongMove_1s04_1_s04_2	:FB_AlarmEvent;
	fbExecLongMove_1s04_2_s05	:FB_AlarmEvent;
	fbExecLongMove_1s05_1s06	:FB_AlarmEvent;
	
//Контроль работы тормозов	
	fbExec_b1K2_b1KM2_err		:FB_AlarmEvent;
	fbExec_b1K3_b1KM3_err		:FB_AlarmEvent;
	fbExec_b1K4_b1KM4_err		:FB_AlarmEvent;
	fbExec_b1K5_b1KM5_err		:FB_AlarmEvent;
	fbExec_b1K6_b1KM6_err		:FB_AlarmEvent;
	fbExec_b1K7_b1KM7_err		:FB_AlarmEvent;
END_VAR

Initialization();
fbButtAlarmReset1_RTRIG (CLK := bButtAlarmReset1);

fbExecAlarm1QF2_1QF7(bAlarmEvent :=bAlarm1QF2_1QF7, bButtAlarmReset:=fbButtAlarmReset1_RTRIG.Q, fbAlarm:=fbAlarm1QF2_1QF7);
fbExecAlarm1QF8(bAlarmEvent :=bAlarm1QF8, bButtAlarmReset:=fbButtAlarmReset1_RTRIG.Q, fbAlarm:=fbAlarm1QF8);
fbExecAlarm1KM2(bAlarmEvent :=bAlarm1KM2, bButtAlarmReset:=fbButtAlarmReset1_RTRIG.Q, fbAlarm:=fbAlarm1KM2);
fbExecAlarm1KM3(bAlarmEvent :=bAlarm1KM3, bButtAlarmReset:=fbButtAlarmReset1_RTRIG.Q, fbAlarm:=fbAlarm1KM3);
fbExecAlarm1KM4(bAlarmEvent :=bAlarm1KM4, bButtAlarmReset:=fbButtAlarmReset1_RTRIG.Q, fbAlarm:=fbAlarm1KM4);
fbExecAlarm1KM5(bAlarmEvent :=bAlarm1KM5, bButtAlarmReset:=fbButtAlarmReset1_RTRIG.Q, fbAlarm:=fbAlarm1KM5);
fbExecAlarm1KM6(bAlarmEvent :=bAlarm1KM6, bButtAlarmReset:=fbButtAlarmReset1_RTRIG.Q, fbAlarm:=fbAlarm1KM6);
fbExecAlarm1KM7(bAlarmEvent :=bAlarm1KM7, bButtAlarmReset:=fbButtAlarmReset1_RTRIG.Q, fbAlarm:=fbAlarm1KM7);

fbExecAlarm_b1_S1_SB0(bAlarmEvent :=bAlarm_b1_S1_SB0, bButtAlarmReset:=fbButtAlarmReset1_RTRIG.Q, fbAlarm:=fbAlarm_b1_S1_SB0);
fbExecAlarm_b1_S6_SB0(bAlarmEvent :=bAlarm_b1_S6_SB0, bButtAlarmReset:=fbButtAlarmReset1_RTRIG.Q, fbAlarm:=fbAlarm_b1_S6_SB0);

fbExecNotDriveReady1s01M1(bAlarmEvent :=bNotDriveReady1s01M1, bButtAlarmReset:=fbButtAlarmReset1_RTRIG.Q, fbAlarm:=fbNotDriveReady1s01M1);
fbExecNotDriveReady1s02M1(bAlarmEvent :=bNotDriveReady1s02M1, bButtAlarmReset:=fbButtAlarmReset1_RTRIG.Q, fbAlarm:=fbNotDriveReady1s02M1);
fbExecNotDriveReady1s03M1(bAlarmEvent :=bNotDriveReady1s03M1, bButtAlarmReset:=fbButtAlarmReset1_RTRIG.Q, fbAlarm:=fbNotDriveReady1s03M1);
fbExecNotDriveReady1s04M1(bAlarmEvent :=bNotDriveReady1s04M1, bButtAlarmReset:=fbButtAlarmReset1_RTRIG.Q, fbAlarm:=fbNotDriveReady1s04M1);
fbExecNotDriveReady1s05M1(bAlarmEvent :=bNotDriveReady1s05M1, bButtAlarmReset:=fbButtAlarmReset1_RTRIG.Q, fbAlarm:=fbNotDriveReady1s05M1);
fbExecNotDriveReady1s06M1(bAlarmEvent :=bNotDriveReady1s06M1, bButtAlarmReset:=fbButtAlarmReset1_RTRIG.Q, fbAlarm:=fbNotDriveReady1s06M1);
(*
fbExecLongMove_1s01_1s02(bAlarmEvent :=bLongMove_1s01_1s02, bButtAlarmReset:=fbButtAlarmReset1_RTRIG.Q, fbAlarm:=fbLongMove_1s01_1s02);
fbExecLongMove_1s02_1s03(bAlarmEvent :=bLongMove_1s02_1s03, bButtAlarmReset:=fbButtAlarmReset1_RTRIG.Q, fbAlarm:=fbLongMove_1s02_1s03);
fbExecLongMove_1s03_1s04(bAlarmEvent :=bLongMove_1s03_1s04, bButtAlarmReset:=fbButtAlarmReset1_RTRIG.Q, fbAlarm:=fbLongMove_1s03_1s04);
fbExecLongMove_1s04_1s05(bAlarmEvent :=bLongMove_1s04_1s05, bButtAlarmReset:=fbButtAlarmReset1_RTRIG.Q, fbAlarm:=fbLongMove_1s04_1s05);
fbExecLongMove_1s05_1s06(bAlarmEvent :=bLongMove_1s05_1s06, bButtAlarmReset:=fbButtAlarmReset1_RTRIG.Q, fbAlarm:=fbLongMove_1s05_1s06);
*)
//тормоза
fbExec_b1K2_b1KM2_err(bAlarmEvent :=b1K2_b1KM2_err, bButtAlarmReset:=fbButtAlarmReset1_RTRIG.Q, fbAlarm:=fbAlarm_b1K2_b1KM2_err);
fbExec_b1K3_b1KM3_err(bAlarmEvent :=b1K3_b1KM3_err, bButtAlarmReset:=fbButtAlarmReset1_RTRIG.Q, fbAlarm:=fbAlarm_b1K3_b1KM3_err);
fbExec_b1K4_b1KM4_err(bAlarmEvent :=b1K4_b1KM4_err, bButtAlarmReset:=fbButtAlarmReset1_RTRIG.Q, fbAlarm:=fbAlarm_b1K4_b1KM4_err);
fbExec_b1K5_b1KM5_err(bAlarmEvent :=b1K5_b1KM5_err, bButtAlarmReset:=fbButtAlarmReset1_RTRIG.Q, fbAlarm:=fbAlarm_b1K5_b1KM5_err);
fbExec_b1K6_b1KM6_err(bAlarmEvent :=b1K6_b1KM6_err, bButtAlarmReset:=fbButtAlarmReset1_RTRIG.Q, fbAlarm:=fbAlarm_b1K6_b1KM6_err);
fbExec_b1K7_b1KM7_err(bAlarmEvent :=b1K7_b1KM7_err, bButtAlarmReset:=fbButtAlarmReset1_RTRIG.Q, fbAlarm:=fbAlarm_b1K7_b1KM7_err);

ACTION Initialization:
IF NOT bIsInitalized THEN
	bIsInitalized := TRUE;
	
	fbAlarm1QF2_1QF7.CreateEx(TC_Events.AlarmConv1.Alarm1QF2_1QF7, TRUE, 0);
	fbAlarm1QF8.CreateEx(TC_Events.AlarmConv1.Alarm1QF8, TRUE, 0);
	fbAlarm1KM2.CreateEx(TC_Events.AlarmConv1.Alarm1KM2, TRUE, 0);
	fbAlarm1KM3.CreateEx(TC_Events.AlarmConv1.Alarm1KM3, TRUE, 0);
	fbAlarm1KM4.CreateEx(TC_Events.AlarmConv1.Alarm1KM4, TRUE, 0);
	fbAlarm1KM5.CreateEx(TC_Events.AlarmConv1.Alarm1KM5, TRUE, 0);
	fbAlarm1KM6.CreateEx(TC_Events.AlarmConv1.Alarm1KM6, TRUE, 0);
	fbAlarm1KM7.CreateEx(TC_Events.AlarmConv1.Alarm1KM7, TRUE, 0);
	
	fbAlarm_b1_S1_SB0.CreateEx(TC_Events.AlarmConv1.Alarm_b1_S1_SB0, TRUE, 0);
	fbAlarm_b1_S6_SB0.CreateEx(TC_Events.AlarmConv1.Alarm_b1_S6_SB0, TRUE, 0);
	
	fbNotDriveReady1s01M1.CreateEx(TC_Events.AlarmConv1.NotDriveReady1s01M1, TRUE, 0);
	fbNotDriveReady1s02M1.CreateEx(TC_Events.AlarmConv1.NotDriveReady1s02M1, TRUE, 0);
	fbNotDriveReady1s03M1.CreateEx(TC_Events.AlarmConv1.NotDriveReady1s03M1, TRUE, 0);
	fbNotDriveReady1s04M1.CreateEx(TC_Events.AlarmConv1.NotDriveReady1s04M1, TRUE, 0);
	fbNotDriveReady1s05M1.CreateEx(TC_Events.AlarmConv1.NotDriveReady1s05M1, TRUE, 0);
	fbNotDriveReady1s06M1.CreateEx(TC_Events.AlarmConv1.NotDriveReady1s06M1, TRUE, 0);
	
	//fbLongMove_1s01_1s02.CreateEx(TC_Events.AlarmConv1.LongMove_1s01_s02_1, TRUE, 0);
	//fbLongMove_1s02_1s03.CreateEx(TC_Events.AlarmConv1.LongMove_1s02_1_s02_2, TRUE, 0);
	//fbLongMove_1s03_1s04.CreateEx(TC_Events.AlarmConv1.LongMove_1s03_1s04, TRUE, 0);
	//fbLongMove_1s04_1s05.CreateEx(TC_Events.AlarmConv1.LongMove_1s04_1s05, TRUE, 0);
	//fbLongMove_1s05_1s06.CreateEx(TC_Events.AlarmConv1.LongMove_1s05_1s06, TRUE, 0);
	fbLongMove_1s01_s02_1.CreateEx(TC_Events.AlarmConv1.LongMove_1s01_s02_1, TRUE, 0);
	fbLongMove_1s01_s02.CreateEx(TC_Events.AlarmConv1.LongMove_1s01_s02, TRUE, 0);
	fbLongMove_1s02_1_s02_2.CreateEx(TC_Events.AlarmConv1.LongMove_1s02_1_s02_2, TRUE, 0);
	fbLongMove_1s02_2_s03_1.CreateEx(TC_Events.AlarmConv1.LongMove_1s02_2_s03_1, TRUE, 0);
	fbLongMove_1s02_s03.CreateEx(TC_Events.AlarmConv1.LongMove_1s01_s02_1, TRUE, 0);
	fbLongMove_1s03_1_s03_2.CreateEx(TC_Events.AlarmConv1.LongMove_1s01_s02_1, TRUE, 0);	
	fbLongMove_1s03_2_s04_1.CreateEx(TC_Events.AlarmConv1.LongMove_1s01_s02_1, TRUE, 0);
	fbLongMove_1s03_s04.CreateEx(TC_Events.AlarmConv1.LongMove_1s01_s02_1, TRUE, 0);	
	fbLongMove_1s04_1_s04_2.CreateEx(TC_Events.AlarmConv1.LongMove_1s01_s02_1, TRUE, 0);
	fbLongMove_1s04_2_s05.CreateEx(TC_Events.AlarmConv1.LongMove_1s01_s02_1, TRUE, 0);
	fbLongMove_1s05_1s06.CreateEx(TC_Events.AlarmConv1.LongMove_1s01_s02_1, TRUE, 0);
	
	//тормоза	
	fbAlarm_b1K2_b1KM2_err.CreateEx(TC_Events.AlarmConv1.Alarm_b1K2_b1KM2_err, TRUE, 0);
	fbAlarm_b1K3_b1KM3_err.CreateEx(TC_Events.AlarmConv1.Alarm_b1K3_b1KM3_err, TRUE, 0);
	fbAlarm_b1K4_b1KM4_err.CreateEx(TC_Events.AlarmConv1.Alarm_b1K4_b1KM4_err, TRUE, 0);
	fbAlarm_b1K5_b1KM5_err.CreateEx(TC_Events.AlarmConv1.Alarm_b1K5_b1KM5_err, TRUE, 0);
	fbAlarm_b1K6_b1KM6_err.CreateEx(TC_Events.AlarmConv1.Alarm_b1K6_b1KM6_err, TRUE, 0);
	fbAlarm_b1K7_b1KM7_err.CreateEx(TC_Events.AlarmConv1.Alarm_b1K7_b1KM7_err, TRUE, 0);
	
END_IF
END_ACTION

END_PROGRAM

// ---- POUs/Alarms/FB_AlarmEvent.TcPOU
FUNCTION_BLOCK FB_AlarmEvent
VAR_INPUT
	bAlarmEvent		:BOOL;
	bButtAlarmReset	:BOOL;
END_VAR
VAR_IN_OUT
	fbAlarm		  :FB_TcAlarm;
END_VAR

IF bAlarmEvent THEN	
	fbAlarm.Raise(0);
END_IF
IF bButtAlarmReset THEN	
	fbAlarm.Clear(0, TRUE);
END_IF

END_FUNCTION_BLOCK

// ---- POUs/Alarms/Alarm_conv_2.TcPOU
PROGRAM Alarm_conv_2
VAR
bAlarm_b2_S1_SB0_blink	:BOOL;
bAlarm_b2_S6_SB0_blink	:BOOL;
Blinking				:BOOL :=TRUE;
END_VAR

//Нет готовности конвейер 2	
	bAlarm2QF2_2QF7 S=NOT b_2QF2_2QF7 	AND bPermAlarm1;
	bAlarm2QF8 		S=NOT b_2QF8 		AND bPermAlarm1;
//	bAlarm2KM2 		S=NOT b_2KM2 		AND bPermAlarm1;
//	bAlarm2KM3 		S=NOT b_2KM3 		AND bPermAlarm1;
//	bAlarm2KM4 		S=NOT b_2KM4 		AND bPermAlarm1;
//	bAlarm2KM5 		S=NOT b_2KM5 		AND bPermAlarm1;
//	bAlarm2KM6 		S=NOT b_2KM6 		AND bPermAlarm1;
//	bAlarm2KM7 		S=NOT b_2KM7 		AND bPermAlarm1;

//Грибки	
	bAlarm_b2_S1_SB0 S=NOT   b2_S1_SB0 	AND bPermAlarm1;
	bAlarm_b2_S6_SB0 S=NOT   b2_S6_SB0 	AND bPermAlarm1;

// Индикация на грибках
	b2S1_SB0 := NOT b2_S1_SB0 AND blink.OUT;
	b2S6_SB0 := NOT b2_S6_SB0 AND blink.OUT;	
	
	blink(ENABLE:=bAlarm_b2_S1_SB0,TIMELOW:=T#500MS,TIMEHIGH:=T#500MS);
	bAlarm_b2_S1_SB0_blink := blink.OUT AND bAlarm_b2_S1_SB0;
	bAlarm_b2_S6_SB0_blink := blink.OUT AND bAlarm_b2_S6_SB0;
	
(*Авария безопасности*)
	bAlarmSafety2 := bAlarm_b2_S1_SB0 OR bAlarm_b2_S6_SB0;

(*Нет общей готовности конвейера 1*)
	bNotReady_2 := bAlarm2QF2_2QF7 OR bAlarm2QF8 OR bAlarm2KM2 OR bAlarm2KM3 OR bAlarm2KM4 OR bAlarm2KM5 OR bAlarm2KM6 OR bAlarm2KM7;

IF  bNotReady2 THEN  sAlarm2:="Нет готовности 2";
		ELSIF bAlarmSafety2 THEN  sAlarm2:="Авария безопасности 2";
			ELSE sAlarm2:="---------";
END_IF

	bPermAlarmDrive2 := bPermAlarm1 AND NOT bAlarmSafety2;

(*(*Готовность *)
	IF NOT bDriveReady2s01M1 AND bPermAlarmDrive2  THEN  bNotDriveReady2s01M1 := TRUE;
	END_IF    
	IF NOT bDriveReady2s02M1 AND bPermAlarmDrive2  THEN  bNotDriveReady2s02M1 := TRUE;
	END_IF 
	IF NOT bDriveReady2s03M1 AND bPermAlarmDrive2  THEN  bNotDriveReady2s03M1 := TRUE;
	END_IF 
	IF NOT bDriveReady2s04M1 AND bPermAlarmDrive2  THEN  bNotDriveReady2s04M1 := TRUE;
	END_IF 
	IF NOT bDriveReady2s05M1 AND bPermAlarmDrive2  THEN  bNotDriveReady2s05M1 := TRUE;
	END_IF 
	IF NOT bDriveReady2s06M1 AND bPermAlarmDrive2  THEN  bNotDriveReady2s06M1 := TRUE;
	END_IF *)

(*Долгие перемещения Drive*)
IF bLongMove2s01_s02_1   THEN bLongMove_2s01_s02_1 := TRUE;
	END_IF
	IF bLongMove2s02_1_s02_2  THEN bLongMove_2s02_1_s02_2 := TRUE;
	END_IF
	IF bLongMove2s02_2_s03_1  THEN bLongMove_2s02_2_s03_1 := TRUE;
	END_IF
	IF bLongMove2s02_s03  THEN bLongMove_2s02_s03 := TRUE;
	END_IF
		IF bLongMove2s03_1_s03_2   THEN bLongMove_2s03_1_s03_2 := TRUE;
	END_IF
	IF bLongMove2s03_2_s04_1  THEN bLongMove_2s03_2_s04_1 := TRUE;
	END_IF
	IF bLongMove2s03_s04  THEN bLongMove_2s03_s04 := TRUE;
	END_IF
	IF bLongMove2s04_1_s04_2  THEN bLongMove_2s04_1_s04_2 := TRUE;
	END_IF
		IF bLongMove2s04_2_s05   THEN bLongMove_2s04_2_s05  := TRUE;
	END_IF
	IF bLongMove2s05_1s06  THEN bLongMove_2s05_1s06 := TRUE;	
	END_IF

(*Нет готовности*)
	bNotReady2 := bNotDriveReady2s01M1 OR bNotDriveReady2s02M1 OR bNotDriveReady2s03M1 OR
			  bNotDriveReady2s04M1 OR bNotDriveReady2s05M1 OR bNotDriveReady2s06M1;

(*Долгое премещение*)
	bLongMove2 := bLongMove_2s02_1_s02_2 OR bLongMove_2s02_1_s02_2  OR bLongMove_2s02_s03 OR
	       bLongMove_2s03_1_s03_2 OR bLongMove_2s03_2_s04_1 OR bLongMove_2s03_s04 OR bLongMove_2s04_1_s04_2 OR
			bLongMove_2s04_2_s05   OR bLongMove_2s05_1s06;

(*Сброс бита аварии по кнопке с панели*)
	bAlarmReset2 := bButtAlarmReset2;

(*Восстановление/сброс аварийных сигналов*)
IF bReset2 OR bAlarmReset2 THEN
	bAlarm2QF8 :=FALSE; bAlarm2QF2_2QF7 :=FALSE; 
	bAlarm2KM2 :=FALSE; bAlarm2KM3 :=FALSE; bAlarm2KM4 :=FALSE; bAlarm2KM5 :=FALSE; bAlarm2KM6 :=FALSE; bAlarm2KM7 :=FALSE;

	bNotDriveReady2s01M1 := FALSE; bNotDriveReady2s02M1 := FALSE; bNotDriveReady2s03M1 := FALSE;
	bNotDriveReady2s04M1 := FALSE; bNotDriveReady2s05M1 := FALSE; bNotDriveReady2s06M1 := FALSE;
	
		bLongMove_2s02_1_s02_2 := FALSE;bLongMove_2s02_1_s02_2 := FALSE; bLongMove_2s02_s03 := FALSE;
	bLongMove_2s03_1_s03_2 := FALSE; bLongMove_2s03_2_s04_1:= FALSE; bLongMove_2s03_s04 := FALSE;
	 bLongMove_2s04_1_s04_2:= FALSE;  bLongMove_2s04_2_s05 := FALSE;
    bLongMove_2s05_1s06 := FALSE;

	bAlarm_b2_S1_SB0 := FALSE; bAlarm_b2_S6_SB0 := FALSE;
END_IF

(*Формирование аварии*)
	bAlarm2 := bNotReady2 OR bLongMove2 OR bAlarmSafety2 OR bNotReady_2 OR bNotReadyGeneral OR bOverflow_CTU_Weight2 OR bOverflow_CTU_ID2;
	bAlarm2_vis := blink.OUT AND bAlarm2;

IF  bNotReady2 THEN  sAlarmLine2:="Нет готовности 2";
		ELSIF bLongMove2 THEN   sAlarmLine2:="Долгое перемещение 2";
			ELSE sAlarmLine2:="---------";
END_IF
IF bAlarm2 THEN bRed_2S1HL1 :=TRUE; bRed_2S1_HL1 := TRUE;
	ELSE bRed_2S1HL1 := FALSE; bRed_2S1_HL1 := FALSE;
END_IF
AlarmEvent_conv2();

END_PROGRAM

// ---- POUs/Alarms/AlarmEvent_conv2.TcPOU
PROGRAM AlarmEvent_conv2
VAR
	bIsInitalized				:BOOL;
	fbButtAlarmReset2_RTRIG 	:R_TRIG;

//готовность конвейера
	fbAlarm2QF2_2QF7			:FB_TcAlarm;
	fbAlarm2QF8					:FB_TcAlarm;
	fbAlarm2KM2					:FB_TcAlarm;
	fbAlarm2KM3					:FB_TcAlarm;
	fbAlarm2KM4					:FB_TcAlarm;
	fbAlarm2KM5					:FB_TcAlarm;
	fbAlarm2KM6					:FB_TcAlarm;
	fbAlarm2KM7					:FB_TcAlarm;
//Грибки	
	fbAlarm_b2_S1_SB0			:FB_TcAlarm;
	fbAlarm_b2_S6_SB0			:FB_TcAlarm;
//готовность двигателей
	fbNotDriveReady2s01M1		:FB_TcAlarm;
	fbNotDriveReady2s02M1		:FB_TcAlarm;
	fbNotDriveReady2s03M1		:FB_TcAlarm;
	fbNotDriveReady2s04M1		:FB_TcAlarm;
	fbNotDriveReady2s05M1		:FB_TcAlarm;
	fbNotDriveReady2s06M1		:FB_TcAlarm;
//Долгие перемещения
	fbLongMove_2s01_2s02		:FB_TcAlarm;
	fbLongMove_2s02_2s03		:FB_TcAlarm;
	fbLongMove_2s03_2s04		:FB_TcAlarm;
	fbLongMove_2s04_2s05		:FB_TcAlarm;
	fbLongMove_2s05_2s06		:FB_TcAlarm;
//----------------------------------------------------------------------------//	
//готовность конвейера
	fbExecAlarm2QF2_2QF7		:FB_AlarmEvent;
	fbExecAlarm2QF8				:FB_AlarmEvent;
	fbExecAlarm2KM2				:FB_AlarmEvent;
	fbExecAlarm2KM3				:FB_AlarmEvent;
	fbExecAlarm2KM4				:FB_AlarmEvent;
	fbExecAlarm2KM5				:FB_AlarmEvent;
	fbExecAlarm2KM6				:FB_AlarmEvent;
	fbExecAlarm2KM7				:FB_AlarmEvent;
//Грибки	
	fbExecAlarm_b2_S1_SB0		:FB_AlarmEvent;
	fbExecAlarm_b2_S6_SB0		:FB_AlarmEvent;
//готовность двигателей
	fbExecNotDriveReady2s01M1	:FB_AlarmEvent;
	fbExecNotDriveReady2s02M1	:FB_AlarmEvent;
	fbExecNotDriveReady2s03M1	:FB_AlarmEvent;
	fbExecNotDriveReady2s04M1	:FB_AlarmEvent;
	fbExecNotDriveReady2s05M1	:FB_AlarmEvent;
	fbExecNotDriveReady2s06M1	:FB_AlarmEvent;
//Долгие перемещения
	fbExecLongMove_2s01_2s02	:FB_AlarmEvent;
	fbExecLongMove_2s02_2s03	:FB_AlarmEvent;
	fbExecLongMove_2s03_2s04	:FB_AlarmEvent;
	fbExecLongMove_2s04_2s05	:FB_AlarmEvent;
	fbExecLongMove_2s05_2s06	:FB_AlarmEvent;	
END_VAR

Initialization();
fbButtAlarmReset2_RTRIG (CLK := bButtAlarmReset2);

fbExecAlarm2QF2_2QF7(bAlarmEvent :=bAlarm2QF2_2QF7, bButtAlarmReset:=fbButtAlarmReset2_RTRIG.Q, fbAlarm:=fbAlarm2QF2_2QF7);
fbExecAlarm2QF8(bAlarmEvent :=bAlarm2QF8, bButtAlarmReset:=fbButtAlarmReset2_RTRIG.Q, fbAlarm:=fbAlarm2QF8);
fbExecAlarm2KM2(bAlarmEvent :=bAlarm2KM2, bButtAlarmReset:=fbButtAlarmReset2_RTRIG.Q, fbAlarm:=fbAlarm2KM2);
fbExecAlarm2KM3(bAlarmEvent :=bAlarm2KM3, bButtAlarmReset:=fbButtAlarmReset2_RTRIG.Q, fbAlarm:=fbAlarm2KM3);
fbExecAlarm2KM4(bAlarmEvent :=bAlarm2KM4, bButtAlarmReset:=fbButtAlarmReset2_RTRIG.Q, fbAlarm:=fbAlarm2KM4);
fbExecAlarm2KM5(bAlarmEvent :=bAlarm2KM5, bButtAlarmReset:=fbButtAlarmReset2_RTRIG.Q, fbAlarm:=fbAlarm2KM5);
fbExecAlarm2KM6(bAlarmEvent :=bAlarm2KM6, bButtAlarmReset:=fbButtAlarmReset2_RTRIG.Q, fbAlarm:=fbAlarm2KM6);
fbExecAlarm2KM7(bAlarmEvent :=bAlarm2KM7, bButtAlarmReset:=fbButtAlarmReset2_RTRIG.Q, fbAlarm:=fbAlarm2KM7);

fbExecAlarm_b2_S1_SB0(bAlarmEvent :=bAlarm_b2_S1_SB0, bButtAlarmReset:=fbButtAlarmReset2_RTRIG.Q, fbAlarm:=fbAlarm_b2_S1_SB0);
fbExecAlarm_b2_S6_SB0(bAlarmEvent :=bAlarm_b2_S6_SB0, bButtAlarmReset:=fbButtAlarmReset2_RTRIG.Q, fbAlarm:=fbAlarm_b2_S6_SB0);

fbExecNotDriveReady2s01M1(bAlarmEvent :=bNotDriveReady2s01M1, bButtAlarmReset:=fbButtAlarmReset2_RTRIG.Q, fbAlarm:=fbNotDriveReady2s01M1);
fbExecNotDriveReady2s02M1(bAlarmEvent :=bNotDriveReady2s02M1, bButtAlarmReset:=fbButtAlarmReset2_RTRIG.Q, fbAlarm:=fbNotDriveReady2s02M1);
fbExecNotDriveReady2s03M1(bAlarmEvent :=bNotDriveReady2s03M1, bButtAlarmReset:=fbButtAlarmReset2_RTRIG.Q, fbAlarm:=fbNotDriveReady2s03M1);
fbExecNotDriveReady2s04M1(bAlarmEvent :=bNotDriveReady2s04M1, bButtAlarmReset:=fbButtAlarmReset2_RTRIG.Q, fbAlarm:=fbNotDriveReady2s04M1);
fbExecNotDriveReady2s05M1(bAlarmEvent :=bNotDriveReady2s05M1, bButtAlarmReset:=fbButtAlarmReset2_RTRIG.Q, fbAlarm:=fbNotDriveReady2s05M1);
fbExecNotDriveReady2s06M1(bAlarmEvent :=bNotDriveReady2s06M1, bButtAlarmReset:=fbButtAlarmReset2_RTRIG.Q, fbAlarm:=fbNotDriveReady2s06M1);

(*fbExecLongMove_2s01_2s02(bAlarmEvent :=bLongMove_2s01_2s02, bButtAlarmReset:=fbButtAlarmReset2_RTRIG.Q, fbAlarm:=fbLongMove_2s01_2s02);
fbExecLongMove_2s02_2s03(bAlarmEvent :=bLongMove_2s02_2s03, bButtAlarmReset:=fbButtAlarmReset2_RTRIG.Q, fbAlarm:=fbLongMove_2s02_2s03);
fbExecLongMove_2s03_2s04(bAlarmEvent :=bLongMove_2s03_2s04, bButtAlarmReset:=fbButtAlarmReset2_RTRIG.Q, fbAlarm:=fbLongMove_2s03_2s04);
fbExecLongMove_2s04_2s05(bAlarmEvent :=bLongMove_2s04_2s05, bButtAlarmReset:=fbButtAlarmReset2_RTRIG.Q, fbAlarm:=fbLongMove_2s04_2s05);
fbExecLongMove_2s05_2s06(bAlarmEvent :=bLongMove_2s05_2s06, bButtAlarmReset:=fbButtAlarmReset2_RTRIG.Q, fbAlarm:=fbLongMove_2s05_2s06);
*)

ACTION Initialization:
IF NOT bIsInitalized THEN
	bIsInitalized := TRUE;
	
	fbAlarm2QF2_2QF7.CreateEx(TC_Events.AlarmConv2.Alarm2QF2_2QF7, TRUE, 0);
	fbAlarm2QF8.CreateEx(TC_Events.AlarmConv2.Alarm2QF8, TRUE, 0);
	fbAlarm2KM2.CreateEx(TC_Events.AlarmConv2.Alarm2KM2, TRUE, 0);
	fbAlarm2KM3.CreateEx(TC_Events.AlarmConv2.Alarm2KM3, TRUE, 0);
	fbAlarm2KM4.CreateEx(TC_Events.AlarmConv2.Alarm2KM4, TRUE, 0);
	fbAlarm2KM5.CreateEx(TC_Events.AlarmConv2.Alarm2KM5, TRUE, 0);
	fbAlarm2KM6.CreateEx(TC_Events.AlarmConv2.Alarm2KM6, TRUE, 0);
	fbAlarm2KM7.CreateEx(TC_Events.AlarmConv2.Alarm2KM7, TRUE, 0);
	
	fbAlarm_b2_S1_SB0.CreateEx(TC_Events.AlarmConv2.Alarm_b2_S1_SB0, TRUE, 0);
	fbAlarm_b2_S6_SB0.CreateEx(TC_Events.AlarmConv2.Alarm_b2_S6_SB0, TRUE, 0);
	
	fbNotDriveReady2s01M1.CreateEx(TC_Events.AlarmConv2.NotDriveReady2s01M1, TRUE, 0);
	fbNotDriveReady2s02M1.CreateEx(TC_Events.AlarmConv2.NotDriveReady2s02M1, TRUE, 0);
	fbNotDriveReady2s03M1.CreateEx(TC_Events.AlarmConv2.NotDriveReady2s03M1, TRUE, 0);
	fbNotDriveReady2s04M1.CreateEx(TC_Events.AlarmConv2.NotDriveReady2s04M1, TRUE, 0);
	fbNotDriveReady2s05M1.CreateEx(TC_Events.AlarmConv2.NotDriveReady2s05M1, TRUE, 0);
	fbNotDriveReady2s06M1.CreateEx(TC_Events.AlarmConv2.NotDriveReady2s06M1, TRUE, 0);
	
	fbLongMove_2s01_2s02.CreateEx(TC_Events.AlarmConv2.LongMove_2s01_2s02, TRUE, 0);
	fbLongMove_2s02_2s03.CreateEx(TC_Events.AlarmConv2.LongMove_2s02_2s03, TRUE, 0);
	fbLongMove_2s03_2s04.CreateEx(TC_Events.AlarmConv2.LongMove_2s03_2s04, TRUE, 0);
	fbLongMove_2s04_2s05.CreateEx(TC_Events.AlarmConv2.LongMove_2s04_2s05, TRUE, 0);
	fbLongMove_2s05_2s06.CreateEx(TC_Events.AlarmConv2.LongMove_2s05_2s06, TRUE, 0);
END_IF
END_ACTION

END_PROGRAM

// ---- POUs/Alarms/Alarm_conv_3.TcPOU
PROGRAM Alarm_conv_3
VAR
bAlarm_b3_S1_SB0_blink	:BOOL;
bAlarm_b3_S6_SB0_blink	:BOOL;
END_VAR

//Нет готовности конвейер 3	
	bAlarm3QF2_3QF7 S=NOT b_3QF2_3QF7 	AND bPermAlarm1;
	bAlarm3QF8 		S=NOT b_3QF8 		AND bPermAlarm1;
//	bAlarm3KM2 		S=NOT b_3KM2 		AND bPermAlarm1;
//	bAlarm3KM3 		S=NOT b_3KM3 		AND bPermAlarm1;
//	bAlarm3KM4 		S=NOT b_3KM4 		AND bPermAlarm1;
//	bAlarm3KM5 		S=NOT b_3KM5 		AND bPermAlarm1;
//	bAlarm3KM6 		S=NOT b_3KM6 		AND bPermAlarm1;
//	bAlarm3KM7 		S=NOT b_3KM7 		AND bPermAlarm1;
	
//Грибки
	bAlarm_b3_S1_SB0 S=NOT   b3_S1_SB0 	AND bPermAlarm1;
	bAlarm_b3_S6_SB0 S=NOT   b3_S6_SB0 	AND bPermAlarm1;

// Индикация на грибках
	b3S1_SB0 := NOT b3_S1_SB0 AND blink.OUT;
	b3S6_SB0 := NOT b3_S6_SB0 AND blink.OUT;	
	
	blink(ENABLE:=bAlarm_b3_S1_SB0,TIMELOW:=T#500MS,TIMEHIGH:=T#500MS);
	bAlarm_b3_S1_SB0_blink := blink.OUT AND bAlarm_b3_S1_SB0;
	bAlarm_b3_S6_SB0_blink := blink.OUT AND bAlarm_b3_S6_SB0;	
(*Авария безопасности*)
	bAlarmSafety3 := bAlarm_b3_S1_SB0 OR bAlarm_b3_S6_SB0;

(*Нет общей готовности конвейера 1*)
	bNotReady_3 := bAlarm3QF2_3QF7 OR bAlarm3QF8 OR bAlarm3KM2 OR bAlarm3KM3 OR bAlarm3KM4 OR bAlarm3KM5 OR bAlarm3KM6 OR bAlarm3KM7;
					
IF  bNotReady3 THEN  sAlarm3:="Нет готовности 3";
		ELSIF bAlarmSafety3 THEN  sAlarm2:="Авария безопасности 3";
			ELSE sAlarm3:="---------";
END_IF

	bPermAlarmDrive3 := bPermAlarm1 AND NOT bAlarmSafety3;

(*(*Готовность *)
	IF NOT bDriveReady3s01M1 AND bPermAlarmDrive3  THEN  bNotDriveReady3s01M1 := TRUE;
	END_IF    
	IF NOT bDriveReady3s02M1 AND bPermAlarmDrive3  THEN  bNotDriveReady3s02M1 := TRUE;
	END_IF 
	IF NOT bDriveReady3s03M1 AND bPermAlarmDrive3  THEN  bNotDriveReady3s03M1 := TRUE;
	END_IF 
	IF NOT bDriveReady3s04M1 AND bPermAlarmDrive3  THEN  bNotDriveReady3s04M1 := TRUE;
	END_IF 
	IF NOT bDriveReady3s05M1 AND bPermAlarmDrive3  THEN  bNotDriveReady3s05M1 := TRUE;
	END_IF 
	IF NOT bDriveReady3s06M1 AND bPermAlarmDrive3  THEN  bNotDriveReady3s06M1 := TRUE;
	END_IF*)

(*Долгие перемещения Drive*)
	IF bLongMove3s01_s02_1   THEN bLongMove_3s01_s02_1 := TRUE;
	END_IF
	IF bLongMove3s02_1_s02_2  THEN bLongMove_3s02_1_s02_2 := TRUE;
	END_IF
	IF bLongMove3s02_2_s03_1  THEN bLongMove_3s02_2_s03_1 := TRUE;
	END_IF
	IF bLongMove3s02_s03  THEN bLongMove_3s02_s03 := TRUE;
	END_IF
		IF bLongMove3s03_1_s03_2   THEN bLongMove_3s03_1_s03_2 := TRUE;
	END_IF
	IF bLongMove3s03_2_s04_1  THEN bLongMove_3s03_2_s04_1 := TRUE;
	END_IF
	IF bLongMove3s03_s04  THEN bLongMove_3s03_s04 := TRUE;
	END_IF
	IF bLongMove3s04_1_s04_2  THEN bLongMove_3s04_1_s04_2 := TRUE;
	END_IF
		IF bLongMove3s04_2_s05   THEN bLongMove_3s04_2_s05  := TRUE;
	END_IF
	IF bLongMove3s05_1s06  THEN bLongMove_3s05_1s06 := TRUE;	
	END_IF
	
(*Нет готовности*)
	bNotReady3 := bNotDriveReady3s01M1 OR bNotDriveReady3s02M1 OR bNotDriveReady3s03M1 OR
			  bNotDriveReady3s04M1 OR bNotDriveReady3s05M1 OR bNotDriveReady3s06M1;

(*Долгое премещение*)
	bLongMove3 :=bLongMove_3s02_1_s02_2 OR bLongMove_3s02_1_s02_2  OR bLongMove_3s02_s03 OR
	       bLongMove_3s03_1_s03_2 OR bLongMove_3s03_2_s04_1 OR bLongMove_3s03_s04 OR bLongMove_3s04_1_s04_2 OR
			bLongMove_3s04_2_s05   OR bLongMove_3s05_1s06;


(*Сброс бита аварии по кнопке с панели*)
	bAlarmReset3 := bButtAlarmReset3;

(*Восстановление/сброс аварийных сигналов*)
IF bReset3 OR bAlarmReset3 THEN
	bAlarm3QF8 :=FALSE; bAlarm3QF2_3QF7 :=FALSE; 
	bAlarm3KM2 :=FALSE; bAlarm3KM3 :=FALSE; bAlarm3KM4 :=FALSE; bAlarm3KM5 :=FALSE; bAlarm3KM6 :=FALSE; bAlarm3KM7 :=FALSE;

	bNotDriveReady3s01M1 := FALSE; bNotDriveReady3s02M1 := FALSE; bNotDriveReady3s03M1 := FALSE;
	bNotDriveReady3s04M1 := FALSE; bNotDriveReady3s05M1 := FALSE; bNotDriveReady3s06M1 := FALSE;
	
	bLongMove_3s02_1_s02_2 := FALSE;bLongMove_3s02_1_s02_2 := FALSE; bLongMove_3s02_s03 := FALSE;
	bLongMove_3s03_1_s03_2 := FALSE; bLongMove_3s03_2_s04_1:= FALSE; bLongMove_3s03_s04 := FALSE;
	 bLongMove_3s04_1_s04_2:= FALSE;  bLongMove_3s04_2_s05 := FALSE;
    bLongMove_3s05_1s06 := FALSE;
	
	
	bAlarm_b3_S1_SB0 := FALSE; bAlarm_b3_S6_SB0 := FALSE;
END_IF

(*Формирование аварии*)
	bAlarm3 := bNotReady3 OR bLongMove3 OR bAlarmSafety3 OR bNotReady_3 OR bNotReadyGeneral OR bOverflow_CTU_Weight3 OR bOverflow_CTU_ID3;
	bAlarm3_vis := blink.OUT AND bAlarm3;
	
IF  bNotReady3 THEN  sAlarmLine3:="Нет готовности 3";
		ELSIF bLongMove3 THEN   sAlarmLine3:="Долгое перемещение 3";
			ELSE sAlarmLine3:="---------";
END_IF
IF bAlarm3 AND b_3AS1 THEN bRed_3S1HL1 :=TRUE; bRed_3S1_HL1 := TRUE;
	ELSE bRed_3S1HL1 := FALSE; bRed_3S1_HL1 := FALSE;
END_IF
AlarmEvent_conv3();

END_PROGRAM

// ---- POUs/Alarms/AlarmEvent_conv3.TcPOU
PROGRAM AlarmEvent_conv3
VAR
	bIsInitalized				:BOOL;
	fbButtAlarmReset3_RTRIG 	:R_TRIG;

//готовность конвейера
	fbAlarm3QF2_3QF7			:FB_TcAlarm;
	fbAlarm3QF8					:FB_TcAlarm;
	fbAlarm3KM2					:FB_TcAlarm;
	fbAlarm3KM3					:FB_TcAlarm;
	fbAlarm3KM4					:FB_TcAlarm;
	fbAlarm3KM5					:FB_TcAlarm;
	fbAlarm3KM6					:FB_TcAlarm;
	fbAlarm3KM7					:FB_TcAlarm;
//Грибки	
	fbAlarm_b3_S1_SB0			:FB_TcAlarm;
	fbAlarm_b3_S6_SB0			:FB_TcAlarm;
//готовность двигателей
	fbNotDriveReady3s01M1		:FB_TcAlarm;
	fbNotDriveReady3s02M1		:FB_TcAlarm;
	fbNotDriveReady3s03M1		:FB_TcAlarm;
	fbNotDriveReady3s04M1		:FB_TcAlarm;
	fbNotDriveReady3s05M1		:FB_TcAlarm;
	fbNotDriveReady3s06M1		:FB_TcAlarm;
//Долгие перемещения
	fbLongMove_3s01_3s02		:FB_TcAlarm;
	fbLongMove_3s02_3s03		:FB_TcAlarm;
	fbLongMove_3s03_3s04		:FB_TcAlarm;
	fbLongMove_3s04_3s05		:FB_TcAlarm;
	fbLongMove_3s05_3s06		:FB_TcAlarm;
//----------------------------------------------------------------------------//	
//готовность конвейера
	fbExecAlarm3QF2_3QF7		:FB_AlarmEvent;
	fbExecAlarm3QF8				:FB_AlarmEvent;
	fbExecAlarm3KM2				:FB_AlarmEvent;
	fbExecAlarm3KM3				:FB_AlarmEvent;
	fbExecAlarm3KM4				:FB_AlarmEvent;
	fbExecAlarm3KM5				:FB_AlarmEvent;
	fbExecAlarm3KM6				:FB_AlarmEvent;
	fbExecAlarm3KM7				:FB_AlarmEvent;
//Грибки	
	fbExecAlarm_b3_S1_SB0		:FB_AlarmEvent;
	fbExecAlarm_b3_S6_SB0		:FB_AlarmEvent;
//готовность двигателей
	fbExecNotDriveReady3s01M1	:FB_AlarmEvent;
	fbExecNotDriveReady3s02M1	:FB_AlarmEvent;
	fbExecNotDriveReady3s03M1	:FB_AlarmEvent;
	fbExecNotDriveReady3s04M1	:FB_AlarmEvent;
	fbExecNotDriveReady3s05M1	:FB_AlarmEvent;
	fbExecNotDriveReady3s06M1	:FB_AlarmEvent;
//Долгие перемещения
	fbExecLongMove_3s01_3s02	:FB_AlarmEvent;
	fbExecLongMove_3s02_3s03	:FB_AlarmEvent;
	fbExecLongMove_3s03_3s04	:FB_AlarmEvent;
	fbExecLongMove_3s04_3s05	:FB_AlarmEvent;
	fbExecLongMove_3s05_3s06	:FB_AlarmEvent;	
END_VAR

Initialization();
fbButtAlarmReset3_RTRIG (CLK := bButtAlarmReset3);

fbExecAlarm3QF2_3QF7(bAlarmEvent :=bAlarm3QF2_3QF7, bButtAlarmReset:=fbButtAlarmReset3_RTRIG.Q, fbAlarm:=fbAlarm3QF2_3QF7);
fbExecAlarm3QF8(bAlarmEvent :=bAlarm3QF8, bButtAlarmReset:=fbButtAlarmReset3_RTRIG.Q, fbAlarm:=fbAlarm3QF8);
fbExecAlarm3KM2(bAlarmEvent :=bAlarm3KM2, bButtAlarmReset:=fbButtAlarmReset3_RTRIG.Q, fbAlarm:=fbAlarm3KM2);
fbExecAlarm3KM3(bAlarmEvent :=bAlarm3KM3, bButtAlarmReset:=fbButtAlarmReset3_RTRIG.Q, fbAlarm:=fbAlarm3KM3);
fbExecAlarm3KM4(bAlarmEvent :=bAlarm3KM4, bButtAlarmReset:=fbButtAlarmReset3_RTRIG.Q, fbAlarm:=fbAlarm3KM4);
fbExecAlarm3KM5(bAlarmEvent :=bAlarm3KM5, bButtAlarmReset:=fbButtAlarmReset3_RTRIG.Q, fbAlarm:=fbAlarm3KM5);
fbExecAlarm3KM6(bAlarmEvent :=bAlarm3KM6, bButtAlarmReset:=fbButtAlarmReset3_RTRIG.Q, fbAlarm:=fbAlarm3KM6);
fbExecAlarm3KM7(bAlarmEvent :=bAlarm3KM7, bButtAlarmReset:=fbButtAlarmReset3_RTRIG.Q, fbAlarm:=fbAlarm3KM7);

fbExecAlarm_b3_S1_SB0(bAlarmEvent :=bAlarm_b3_S1_SB0, bButtAlarmReset:=fbButtAlarmReset3_RTRIG.Q, fbAlarm:=fbAlarm_b3_S1_SB0);
fbExecAlarm_b3_S6_SB0(bAlarmEvent :=bAlarm_b3_S6_SB0, bButtAlarmReset:=fbButtAlarmReset3_RTRIG.Q, fbAlarm:=fbAlarm_b3_S6_SB0);

fbExecNotDriveReady3s01M1(bAlarmEvent :=bNotDriveReady3s01M1, bButtAlarmReset:=fbButtAlarmReset3_RTRIG.Q, fbAlarm:=fbNotDriveReady3s01M1);
fbExecNotDriveReady3s02M1(bAlarmEvent :=bNotDriveReady3s02M1, bButtAlarmReset:=fbButtAlarmReset3_RTRIG.Q, fbAlarm:=fbNotDriveReady3s02M1);
fbExecNotDriveReady3s03M1(bAlarmEvent :=bNotDriveReady3s03M1, bButtAlarmReset:=fbButtAlarmReset3_RTRIG.Q, fbAlarm:=fbNotDriveReady3s03M1);
fbExecNotDriveReady3s04M1(bAlarmEvent :=bNotDriveReady3s04M1, bButtAlarmReset:=fbButtAlarmReset3_RTRIG.Q, fbAlarm:=fbNotDriveReady3s04M1);
fbExecNotDriveReady3s05M1(bAlarmEvent :=bNotDriveReady3s05M1, bButtAlarmReset:=fbButtAlarmReset3_RTRIG.Q, fbAlarm:=fbNotDriveReady3s05M1);
fbExecNotDriveReady3s06M1(bAlarmEvent :=bNotDriveReady3s06M1, bButtAlarmReset:=fbButtAlarmReset3_RTRIG.Q, fbAlarm:=fbNotDriveReady3s06M1);

(*fbExecLongMove_3s01_3s02(bAlarmEvent :=bLongMove_3s01_3s02, bButtAlarmReset:=fbButtAlarmReset3_RTRIG.Q, fbAlarm:=fbLongMove_3s01_3s02);
fbExecLongMove_3s02_3s03(bAlarmEvent :=bLongMove_3s02_3s03, bButtAlarmReset:=fbButtAlarmReset3_RTRIG.Q, fbAlarm:=fbLongMove_3s02_3s03);
fbExecLongMove_3s03_3s04(bAlarmEvent :=bLongMove_3s03_3s04, bButtAlarmReset:=fbButtAlarmReset3_RTRIG.Q, fbAlarm:=fbLongMove_3s03_3s04);
fbExecLongMove_3s04_3s05(bAlarmEvent :=bLongMove_3s04_3s05, bButtAlarmReset:=fbButtAlarmReset3_RTRIG.Q, fbAlarm:=fbLongMove_3s04_3s05);
fbExecLongMove_3s05_3s06(bAlarmEvent :=bLongMove_3s05_3s06, bButtAlarmReset:=fbButtAlarmReset3_RTRIG.Q, fbAlarm:=fbLongMove_3s05_3s06);
*)

ACTION Initialization:
IF NOT bIsInitalized THEN
	bIsInitalized := TRUE;
	
	fbAlarm3QF2_3QF7.CreateEx(TC_Events.AlarmConv3.Alarm3QF2_3QF7, TRUE, 0);
	fbAlarm3QF8.CreateEx(TC_Events.AlarmConv3.Alarm3QF8, TRUE, 0);
	fbAlarm3KM2.CreateEx(TC_Events.AlarmConv3.Alarm3KM2, TRUE, 0);
	fbAlarm3KM3.CreateEx(TC_Events.AlarmConv3.Alarm3KM3, TRUE, 0);
	fbAlarm3KM4.CreateEx(TC_Events.AlarmConv3.Alarm3KM4, TRUE, 0);
	fbAlarm3KM5.CreateEx(TC_Events.AlarmConv3.Alarm3KM5, TRUE, 0);
	fbAlarm3KM6.CreateEx(TC_Events.AlarmConv3.Alarm3KM6, TRUE, 0);
	fbAlarm3KM7.CreateEx(TC_Events.AlarmConv3.Alarm3KM7, TRUE, 0);
	
	fbAlarm_b3_S1_SB0.CreateEx(TC_Events.AlarmConv3.Alarm_b3_S1_SB0, TRUE, 0);
	fbAlarm_b3_S6_SB0.CreateEx(TC_Events.AlarmConv3.Alarm_b3_S6_SB0, TRUE, 0);
	
	fbNotDriveReady3s01M1.CreateEx(TC_Events.AlarmConv3.NotDriveReady3s01M1, TRUE, 0);
	fbNotDriveReady3s02M1.CreateEx(TC_Events.AlarmConv3.NotDriveReady3s02M1, TRUE, 0);
	fbNotDriveReady3s03M1.CreateEx(TC_Events.AlarmConv3.NotDriveReady3s03M1, TRUE, 0);
	fbNotDriveReady3s04M1.CreateEx(TC_Events.AlarmConv3.NotDriveReady3s04M1, TRUE, 0);
	fbNotDriveReady3s05M1.CreateEx(TC_Events.AlarmConv3.NotDriveReady3s05M1, TRUE, 0);
	fbNotDriveReady3s06M1.CreateEx(TC_Events.AlarmConv3.NotDriveReady3s06M1, TRUE, 0);
	
	fbLongMove_3s01_3s02.CreateEx(TC_Events.AlarmConv3.LongMove_3s01_3s02, TRUE, 0);
	fbLongMove_3s02_3s03.CreateEx(TC_Events.AlarmConv3.LongMove_3s02_3s03, TRUE, 0);
	fbLongMove_3s03_3s04.CreateEx(TC_Events.AlarmConv3.LongMove_3s03_3s04, TRUE, 0);
	fbLongMove_3s04_3s05.CreateEx(TC_Events.AlarmConv3.LongMove_3s04_3s05, TRUE, 0);
	fbLongMove_3s05_3s06.CreateEx(TC_Events.AlarmConv3.LongMove_3s05_3s06, TRUE, 0);
END_IF
END_ACTION

END_PROGRAM

// ---- POUs/Alarms/Alarm_conv_4.TcPOU
PROGRAM Alarm_conv_4
VAR
bAlarm_b4_S1_SB0_blink	:BOOL;
bAlarm_b4_S6_SB0_blink	:BOOL;
END_VAR

//Нет готовности конвейер 4	
	bAlarm4QF2_4QF7 S=NOT b_4QF2_4QF7 	AND bPermAlarm1;
	bAlarm4QF8 		S=NOT b_4QF8 		AND bPermAlarm1;
//	bAlarm4KM2 		S=NOT b_4KM2 		AND bPermAlarm1;
//	bAlarm4KM3 		S=NOT b_4KM3 		AND bPermAlarm1;
//	bAlarm4KM4 		S=NOT b_4KM4 		AND bPermAlarm1;
//	bAlarm4KM5 		S=NOT b_4KM5 		AND bPermAlarm1;
//	bAlarm4KM6 		S=NOT b_4KM6 		AND bPermAlarm1;
//	bAlarm4KM7 		S=NOT b_4KM7 		AND bPermAlarm1;
	
//Грибки
	bAlarm_b4_S1_SB0 S=NOT   b4_S1_SB0 	AND bPermAlarm1;
	bAlarm_b4_S6_SB0 S=NOT   b4_S6_SB0  	AND bPermAlarm1;

// Индикация на грибках
	b4S1_SB0 := NOT b4_S1_SB0 AND blink.OUT;
	b4S6_SB0 := NOT b4_S6_SB0 AND blink.OUT;	
	
	blink(ENABLE:=bAlarm_b4_S1_SB0,TIMELOW:=T#500MS,TIMEHIGH:=T#500MS);
	bAlarm_b4_S1_SB0_blink := NOT blink.OUT AND bAlarm_b4_S1_SB0;
	bAlarm_b4_S6_SB0_blink := NOT blink.OUT AND bAlarm_b4_S6_SB0;	
(*Авария безопасности*)
	bAlarmSafety4 := bAlarm_b4_S1_SB0 OR bAlarm_b4_S6_SB0;

(*Нет общей готовности конвейера 1*)
	bNotReady_4 := bAlarm4QF2_4QF7 OR bAlarm4QF8 OR bAlarm4KM2 OR bAlarm4KM3 OR bAlarm4KM4 OR bAlarm4KM5 OR bAlarm4KM6 OR bAlarm4KM7;

IF  bNotReady4 THEN  sAlarm4:="Нет готовности 4";
		ELSIF bAlarmSafety4 THEN  sAlarm4:="Авария безопасности 4";
			ELSE sAlarm4:="---------";
END_IF

	bPermAlarmDrive4 := bPermAlarm1 AND NOT bAlarmSafety4;

(*(*Готовность *)
	IF NOT bDriveReady4s01M1 AND bPermAlarmDrive4  THEN  bNotDriveReady4s01M1 := TRUE;
	END_IF    
	IF NOT bDriveReady4s02M1 AND bPermAlarmDrive4  THEN  bNotDriveReady4s02M1 := TRUE;
	END_IF 
	IF NOT bDriveReady4s03M1 AND bPermAlarmDrive4  THEN  bNotDriveReady4s03M1 := TRUE;
	END_IF 
	IF NOT bDriveReady4s04M1 AND bPermAlarmDrive4  THEN  bNotDriveReady4s04M1 := TRUE;
	END_IF 
	IF NOT bDriveReady4s05M1 AND bPermAlarmDrive4  THEN  bNotDriveReady4s05M1 := TRUE;
	END_IF 
	IF NOT bDriveReady4s06M1 AND bPermAlarmDrive4  THEN  bNotDriveReady4s06M1 := TRUE;
	END_IF *)

(*Долгие перемещения Drive*)
	IF bLongMove4s01_s02_1   THEN bLongMove_4s01_s02_1 := TRUE;
	END_IF
	IF bLongMove4s02_1_s02_2  THEN bLongMove_4s02_1_s02_2 := TRUE;
	END_IF
	IF bLongMove4s02_2_s03_1  THEN bLongMove_4s02_2_s03_1 := TRUE;
	END_IF
	IF bLongMove4s02_s03  THEN bLongMove_4s02_s03 := TRUE;
	END_IF
		IF bLongMove4s03_1_s03_2   THEN bLongMove_4s03_1_s03_2 := TRUE;
	END_IF
	IF bLongMove4s03_2_s04_1  THEN bLongMove_4s03_2_s04_1 := TRUE;
	END_IF
	IF bLongMove4s03_s04  THEN bLongMove_4s03_s04 := TRUE;
	END_IF
	IF bLongMove4s04_1_s04_2  THEN bLongMove_4s04_1_s04_2 := TRUE;
	END_IF
		IF bLongMove4s04_2_s05   THEN bLongMove_4s04_2_s05  := TRUE;
	END_IF
	IF bLongMove4s05_1s06  THEN bLongMove_4s05_1s06 := TRUE;	
	END_IF
(*Нет готовности*)
	bNotReady4 := bNotDriveReady4s01M1 OR bNotDriveReady4s02M1 OR bNotDriveReady4s03M1 OR
			  bNotDriveReady4s04M1 OR bNotDriveReady4s05M1 OR bNotDriveReady4s06M1;

(*Долгое премещение*)
	bLongMove4 := bLongMove_4s02_1_s02_2 OR bLongMove_4s02_1_s02_2  OR bLongMove_4s02_s03 OR
	       bLongMove_4s03_1_s03_2 OR bLongMove_4s03_2_s04_1 OR bLongMove_4s03_s04 OR bLongMove_4s04_1_s04_2 OR
			bLongMove_4s04_2_s05   OR bLongMove_4s05_1s06;

(*Сброс бита аварии по кнопке с панели*)
	bAlarmReset4 := bButtAlarmReset4;

(*Восстановление/сброс аварийных сигналов*)
IF bReset4 OR bAlarmReset4 THEN
	bAlarm4QF8 :=FALSE; bAlarm4QF2_4QF7 :=FALSE; 
	bAlarm4KM2 :=FALSE; bAlarm4KM3 :=FALSE; bAlarm4KM4 :=FALSE; bAlarm4KM5 :=FALSE; bAlarm4KM6 :=FALSE; bAlarm4KM7 :=FALSE;

	bNotDriveReady4s01M1 := FALSE; bNotDriveReady4s02M1 := FALSE; bNotDriveReady4s03M1 := FALSE;
	bNotDriveReady4s04M1 := FALSE; bNotDriveReady4s05M1 := FALSE; bNotDriveReady4s06M1 := FALSE;
	
	bLongMove_4s02_1_s02_2 := FALSE;bLongMove_4s02_1_s02_2 := FALSE; bLongMove_4s02_s03 := FALSE;
	bLongMove_4s03_1_s03_2 := FALSE; bLongMove_4s03_2_s04_1:= FALSE; bLongMove_4s03_s04 := FALSE;
	 bLongMove_4s04_1_s04_2:= FALSE;  bLongMove_4s04_2_s05 := FALSE;
    bLongMove_4s05_1s06 := FALSE;
	
	
	bAlarm_b4_S1_SB0 := FALSE; bAlarm_b4_S6_SB0 := FALSE;
END_IF

(*Формирование аварии*)
	bAlarm4 := bNotReady4 OR bLongMove4 OR bAlarmSafety4 OR bNotReady_4 OR bNotReadyGeneral OR bOverflow_CTU_Weight4 OR bOverflow_CTU_ID4;
	bAlarm4_vis := blink.OUT AND bAlarm4;
IF  bNotReady4 THEN  sAlarmLine4:="Нет готовности 4";
		ELSIF bLongMove4 THEN   sAlarmLine4:="Долгое перемещение 4";
			ELSE sAlarmLine4:="---------";
END_IF
IF bAlarm4 AND b_4AS1 THEN bRed_4S1HL1 :=TRUE; bRed_4S1_HL1 := TRUE;
	ELSE bRed_4S1HL1 := FALSE; bRed_4S1_HL1 := FALSE;
END_IF
AlarmEvent_conv4();

END_PROGRAM

// ---- POUs/Alarms/AlarmEvent_conv4.TcPOU
PROGRAM AlarmEvent_conv4
VAR
	bIsInitalized				:BOOL;
	fbButtAlarmReset4_RTRIG 	:R_TRIG;

//готовность конвейера
	fbAlarm4QF2_4QF7			:FB_TcAlarm;
	fbAlarm4QF8					:FB_TcAlarm;
	fbAlarm4KM2					:FB_TcAlarm;
	fbAlarm4KM3					:FB_TcAlarm;
	fbAlarm4KM4					:FB_TcAlarm;
	fbAlarm4KM5					:FB_TcAlarm;
	fbAlarm4KM6					:FB_TcAlarm;
	fbAlarm4KM7					:FB_TcAlarm;
//Грибки	
	fbAlarm_b4_S1_SB0			:FB_TcAlarm;
	fbAlarm_b4_S6_SB0			:FB_TcAlarm;
//готовность двигателей
	fbNotDriveReady4s01M1		:FB_TcAlarm;
	fbNotDriveReady4s02M1		:FB_TcAlarm;
	fbNotDriveReady4s03M1		:FB_TcAlarm;
	fbNotDriveReady4s04M1		:FB_TcAlarm;
	fbNotDriveReady4s05M1		:FB_TcAlarm;
	fbNotDriveReady4s06M1		:FB_TcAlarm;
//Долгие перемещения
	fbLongMove_4s01_4s02		:FB_TcAlarm;
	fbLongMove_4s02_4s03		:FB_TcAlarm;
	fbLongMove_4s03_4s04		:FB_TcAlarm;
	fbLongMove_4s04_4s05		:FB_TcAlarm;
	fbLongMove_4s05_4s06		:FB_TcAlarm;
//----------------------------------------------------------------------------//	
//готовность конвейера
	fbExecAlarm4QF2_4QF7		:FB_AlarmEvent;
	fbExecAlarm4QF8				:FB_AlarmEvent;
	fbExecAlarm4KM2				:FB_AlarmEvent;
	fbExecAlarm4KM3				:FB_AlarmEvent;
	fbExecAlarm4KM4				:FB_AlarmEvent;
	fbExecAlarm4KM5				:FB_AlarmEvent;
	fbExecAlarm4KM6				:FB_AlarmEvent;
	fbExecAlarm4KM7				:FB_AlarmEvent;
//Грибки	
	fbExecAlarm_b4_S1_SB0		:FB_AlarmEvent;
	fbExecAlarm_b4_S6_SB0		:FB_AlarmEvent;
//готовность двигателей
	fbExecNotDriveReady4s01M1	:FB_AlarmEvent;
	fbExecNotDriveReady4s02M1	:FB_AlarmEvent;
	fbExecNotDriveReady4s03M1	:FB_AlarmEvent;
	fbExecNotDriveReady4s04M1	:FB_AlarmEvent;
	fbExecNotDriveReady4s05M1	:FB_AlarmEvent;
	fbExecNotDriveReady4s06M1	:FB_AlarmEvent;
//Долгие перемещения
	fbExecLongMove_4s01_4s02	:FB_AlarmEvent;
	fbExecLongMove_4s02_4s03	:FB_AlarmEvent;
	fbExecLongMove_4s03_4s04	:FB_AlarmEvent;
	fbExecLongMove_4s04_4s05	:FB_AlarmEvent;
	fbExecLongMove_4s05_4s06	:FB_AlarmEvent;	
END_VAR

Initialization();
fbButtAlarmReset4_RTRIG (CLK := bButtAlarmReset4);

fbExecAlarm4QF2_4QF7(bAlarmEvent :=bAlarm4QF2_4QF7, bButtAlarmReset:=fbButtAlarmReset4_RTRIG.Q, fbAlarm:=fbAlarm4QF2_4QF7);
fbExecAlarm4QF8(bAlarmEvent :=bAlarm4QF8, bButtAlarmReset:=fbButtAlarmReset4_RTRIG.Q, fbAlarm:=fbAlarm4QF8);
fbExecAlarm4KM2(bAlarmEvent :=bAlarm4KM2, bButtAlarmReset:=fbButtAlarmReset4_RTRIG.Q, fbAlarm:=fbAlarm4KM2);
fbExecAlarm4KM3(bAlarmEvent :=bAlarm4KM3, bButtAlarmReset:=fbButtAlarmReset4_RTRIG.Q, fbAlarm:=fbAlarm4KM3);
fbExecAlarm4KM4(bAlarmEvent :=bAlarm4KM4, bButtAlarmReset:=fbButtAlarmReset4_RTRIG.Q, fbAlarm:=fbAlarm4KM4);
fbExecAlarm4KM5(bAlarmEvent :=bAlarm4KM5, bButtAlarmReset:=fbButtAlarmReset4_RTRIG.Q, fbAlarm:=fbAlarm4KM5);
fbExecAlarm4KM6(bAlarmEvent :=bAlarm4KM6, bButtAlarmReset:=fbButtAlarmReset4_RTRIG.Q, fbAlarm:=fbAlarm4KM6);
fbExecAlarm4KM7(bAlarmEvent :=bAlarm4KM7, bButtAlarmReset:=fbButtAlarmReset4_RTRIG.Q, fbAlarm:=fbAlarm4KM7);

fbExecAlarm_b4_S1_SB0(bAlarmEvent :=bAlarm_b4_S1_SB0, bButtAlarmReset:=fbButtAlarmReset4_RTRIG.Q, fbAlarm:=fbAlarm_b4_S1_SB0);
fbExecAlarm_b4_S6_SB0(bAlarmEvent :=bAlarm_b4_S6_SB0, bButtAlarmReset:=fbButtAlarmReset4_RTRIG.Q, fbAlarm:=fbAlarm_b4_S6_SB0);

fbExecNotDriveReady4s01M1(bAlarmEvent :=bNotDriveReady4s01M1, bButtAlarmReset:=fbButtAlarmReset4_RTRIG.Q, fbAlarm:=fbNotDriveReady4s01M1);
fbExecNotDriveReady4s02M1(bAlarmEvent :=bNotDriveReady4s02M1, bButtAlarmReset:=fbButtAlarmReset4_RTRIG.Q, fbAlarm:=fbNotDriveReady4s02M1);
fbExecNotDriveReady4s03M1(bAlarmEvent :=bNotDriveReady4s03M1, bButtAlarmReset:=fbButtAlarmReset4_RTRIG.Q, fbAlarm:=fbNotDriveReady4s03M1);
fbExecNotDriveReady4s04M1(bAlarmEvent :=bNotDriveReady4s04M1, bButtAlarmReset:=fbButtAlarmReset4_RTRIG.Q, fbAlarm:=fbNotDriveReady4s04M1);
fbExecNotDriveReady4s05M1(bAlarmEvent :=bNotDriveReady4s05M1, bButtAlarmReset:=fbButtAlarmReset4_RTRIG.Q, fbAlarm:=fbNotDriveReady4s05M1);
fbExecNotDriveReady4s06M1(bAlarmEvent :=bNotDriveReady4s06M1, bButtAlarmReset:=fbButtAlarmReset4_RTRIG.Q, fbAlarm:=fbNotDriveReady4s06M1);

(*fbExecLongMove_4s01_4s02(bAlarmEvent :=bLongMove_4s01_4s02, bButtAlarmReset:=fbButtAlarmReset4_RTRIG.Q, fbAlarm:=fbLongMove_4s01_4s02);
fbExecLongMove_4s02_4s03(bAlarmEvent :=bLongMove_4s02_4s03, bButtAlarmReset:=fbButtAlarmReset4_RTRIG.Q, fbAlarm:=fbLongMove_4s02_4s03);
fbExecLongMove_4s03_4s04(bAlarmEvent :=bLongMove_4s03_4s04, bButtAlarmReset:=fbButtAlarmReset4_RTRIG.Q, fbAlarm:=fbLongMove_4s03_4s04);
fbExecLongMove_4s04_4s05(bAlarmEvent :=bLongMove_4s04_4s05, bButtAlarmReset:=fbButtAlarmReset4_RTRIG.Q, fbAlarm:=fbLongMove_4s04_4s05);
fbExecLongMove_4s05_4s06(bAlarmEvent :=bLongMove_4s05_4s06, bButtAlarmReset:=fbButtAlarmReset4_RTRIG.Q, fbAlarm:=fbLongMove_4s05_4s06);
*)

ACTION Initialization:
IF NOT bIsInitalized THEN
	bIsInitalized := TRUE;
	
	fbAlarm4QF2_4QF7.CreateEx(TC_Events.AlarmConv4.Alarm4QF2_4QF7, TRUE, 0);
	fbAlarm4QF8.CreateEx(TC_Events.AlarmConv4.Alarm4QF8, TRUE, 0);
	fbAlarm4KM2.CreateEx(TC_Events.AlarmConv4.Alarm4KM2, TRUE, 0);
	fbAlarm4KM3.CreateEx(TC_Events.AlarmConv4.Alarm4KM3, TRUE, 0);
	fbAlarm4KM4.CreateEx(TC_Events.AlarmConv4.Alarm4KM4, TRUE, 0);
	fbAlarm4KM5.CreateEx(TC_Events.AlarmConv4.Alarm4KM5, TRUE, 0);
	fbAlarm4KM6.CreateEx(TC_Events.AlarmConv4.Alarm4KM6, TRUE, 0);
	fbAlarm4KM7.CreateEx(TC_Events.AlarmConv4.Alarm4KM7, TRUE, 0);
	
	fbAlarm_b4_S1_SB0.CreateEx(TC_Events.AlarmConv4.Alarm_b4_S1_SB0, TRUE, 0);
	fbAlarm_b4_S6_SB0.CreateEx(TC_Events.AlarmConv4.Alarm_b4_S6_SB0, TRUE, 0);
	
	fbNotDriveReady4s01M1.CreateEx(TC_Events.AlarmConv4.NotDriveReady4s01M1, TRUE, 0);
	fbNotDriveReady4s02M1.CreateEx(TC_Events.AlarmConv4.NotDriveReady4s02M1, TRUE, 0);
	fbNotDriveReady4s03M1.CreateEx(TC_Events.AlarmConv4.NotDriveReady4s03M1, TRUE, 0);
	fbNotDriveReady4s04M1.CreateEx(TC_Events.AlarmConv4.NotDriveReady4s04M1, TRUE, 0);
	fbNotDriveReady4s05M1.CreateEx(TC_Events.AlarmConv4.NotDriveReady4s05M1, TRUE, 0);
	fbNotDriveReady4s06M1.CreateEx(TC_Events.AlarmConv4.NotDriveReady4s06M1, TRUE, 0);
	
	fbLongMove_4s01_4s02.CreateEx(TC_Events.AlarmConv4.LongMove_4s01_4s02, TRUE, 0);
	fbLongMove_4s02_4s03.CreateEx(TC_Events.AlarmConv4.LongMove_4s02_4s03, TRUE, 0);
	fbLongMove_4s03_4s04.CreateEx(TC_Events.AlarmConv4.LongMove_4s03_4s04, TRUE, 0);
	fbLongMove_4s04_4s05.CreateEx(TC_Events.AlarmConv4.LongMove_4s04_4s05, TRUE, 0);
	fbLongMove_4s05_4s06.CreateEx(TC_Events.AlarmConv4.LongMove_4s05_4s06, TRUE, 0);
END_IF
END_ACTION

END_PROGRAM

// ---- POUs/Alarms/Alarm_conv_General.TcPOU
	PROGRAM Alarm_conv_General
VAR
Blink_All1	:BLINK;
Blink_All2	:BLINK;
start		:BOOL := TRUE;
ReadyOK1 	:BOOL;
ReadyOK2 	:BOOL;
ReadyOK3 	:BOOL;
ReadyOK4 	:BOOL;

fbDirection1:FB_Direction;
fbDirection2:FB_Direction;
fbDirection3:FB_Direction;
fbDirection4:FB_Direction;

END_VAR

Blink_All1(ENABLE := start, TIMELOW := T#1000MS, TIMEHIGH :=T#500MS);
Blink_All2(ENABLE := start, TIMELOW := T#500MS, TIMEHIGH :=T#500MS);

//Нет готовности блоков питания
	bNotReadyPower24v 	S=NOT b_GP3;
  	bPermAlarm1			:=NOT bNotReadyPower24v;

//УЗИП
	bAlarm1QF 			S=NOT b_1QF  AND bPermAlarm1;
	bAlarm2QF 			S=NOT b_2QF  AND bPermAlarm1;

	bAlarmQF := bAlarm1QF OR bAlarm2QF;
	
//Вспомогательные системы
	bAlarmSF3 			S=NOT b_SF3  AND bPermAlarm1;
	bAlarmSF3_ 			S=NOT b_SF3_ AND bPermAlarm1;
	
	bAlarmSF := bAlarmSF3 OR bAlarmSF3_;

//Аварии ввода	
	bAlarmK2 			S=NOT b_K2   AND bPermAlarm1;
	bAlarmK2_ 			S=NOT b_K2_  AND bPermAlarm1;
	
	bAlarm_Input_accident := bAlarmK2 OR bAlarmK2_;	
	
//Реле безопасности	
	bAlarm1AS1 			S= NOT b_1AS1 AND bPermAlarm1;
	bAlarm2AS1 			S= NOT b_2AS1 AND bPermAlarm1;
	bAlarm3AS1 			S= NOT b_3AS1 AND bPermAlarm1;	
	bAlarm4AS1 			S= NOT b_4AS1 AND bPermAlarm1;
	
	bAlarm_Safety_relay := bAlarm1AS1 OR bAlarm2AS1 OR 
						   bAlarm3AS1 OR bAlarm4AS1;
	
//Питание приводов	
	bAlarm1QF1 			S=NOT b_1QF1 AND bPermAlarm1;
	bAlarm2QF1 			S=NOT b_2QF1 AND bPermAlarm1;
	bAlarm3QF1 			S=NOT b_3QF1 AND bPermAlarm1;
	bAlarm4QF1 			S=NOT b_4QF1 AND bPermAlarm1;
	
	bAlarm_Drive_power := bAlarm1QF1 OR bAlarm2QF1 OR 
						  bAlarm3QF1 OR bAlarm4QF1;

//Превышение тока или напряжения
//	bAlarm1P_I 			S=NOT b_1P_I AND bPermAlarm1;
//	bAlarm1P_U 			S=NOT b_1P_U AND bPermAlarm1;

	bAlarm_Overload_I_U := bAlarm1P_I OR bAlarm1P_U;

(*Нет общей готовности*)
	bNotReadyGeneral := bNotReadyPower24v OR bAlarmQF OR bAlarmSF OR 
						bAlarm_Input_accident OR bAlarm_Safety_relay OR 
						bAlarm_Drive_power OR bAlarm_Overload_I_U;

IF bButtAlarmResetGeneral THEN 
	bNotReadyPower24v :=FALSE; 
	bAlarmK2 :=FALSE; bAlarmK2_ :=FALSE;	
	bAlarm1QF :=FALSE; bAlarm2QF :=FALSE; 
	bAlarmSF3 :=FALSE; bAlarmSF3_ :=FALSE; 	
	bAlarm1P_I :=FALSE; bAlarm1P_U :=FALSE;
	bAlarm1AS1 :=FALSE; bAlarm2AS1 :=FALSE; bAlarm3AS1 :=FALSE; bAlarm4AS1 :=FALSE; 
	bAlarm1QF1 :=FALSE; bAlarm2QF1 :=FALSE; bAlarm3QF1 :=FALSE; bAlarm4QF1 :=FALSE; 
	bAlarm1QF8 :=FALSE; bAlarm2QF8 :=FALSE; bAlarm3QF8 :=FALSE; bAlarm4QF8 :=FALSE; 
	bAlarm1QF2_1QF7 :=FALSE; bAlarm2QF2_2QF7 :=FALSE; bAlarm3QF2_3QF7 :=FALSE; bAlarm4QF2_4QF7 :=FALSE; 
	bAlarm1KM2 :=FALSE; bAlarm1KM3 :=FALSE; bAlarm1KM4 :=FALSE; bAlarm1KM5 :=FALSE; bAlarm1KM6 :=FALSE; bAlarm1KM7 :=FALSE;
	bAlarm2KM2 :=FALSE; bAlarm2KM3 :=FALSE; bAlarm2KM4 :=FALSE; bAlarm2KM5 :=FALSE; bAlarm2KM6 :=FALSE; bAlarm2KM7 :=FALSE;
	bAlarm3KM2 :=FALSE; bAlarm3KM3 :=FALSE; bAlarm3KM4 :=FALSE; bAlarm3KM5 :=FALSE; bAlarm3KM6 :=FALSE; bAlarm3KM7 :=FALSE;
	bAlarm4KM2 :=FALSE; bAlarm4KM3 :=FALSE; bAlarm4KM4 :=FALSE; bAlarm4KM5 :=FALSE; bAlarm4KM6 :=FALSE; bAlarm4KM7 :=FALSE;
END_IF

b1Sh_SB1 := NOT bAlarm1 AND NOT bAlarm2 AND NOT bNotReadyGeneral AND Blink_All1.OUT AND NOT b_1AS1 AND NOT b_2AS1;
b2Sh_SB1 := NOT bAlarm3 AND NOT bAlarm4 AND NOT bNotReadyGeneral AND Blink_All1.OUT AND NOT b_3AS1 AND NOT b_4AS1;

ReadyOK1 := NOT bAlarm1 AND NOT bNotReadyGeneral AND b_1AS1; 
//b_1K1_1 := ReadyOK1 AND NOT b_1KM1_2  (*bButtReverse1*) AND (bAutomat1 OR bManual1) AND NOT bReverse1;
ReadyOK2 := NOT bAlarm2 AND NOT bNotReadyGeneral AND b_2AS1; 
//b_2K1_1 := ReadyOK2 AND NOT bButtReverse2 AND (bAutomat2 OR bManual2) AND NOT bReverse2;
ReadyOK3 := NOT bAlarm3 AND NOT bNotReadyGeneral AND b_3AS1; 
//b_3K1_1 := ReadyOK3 AND NOT bButtReverse3 AND (bAutomat3 OR bManual3) AND NOT bReverse3;
ReadyOK4 := NOT bAlarm4 AND NOT bNotReadyGeneral AND b_4AS1; 
//b_4K1_1 := ReadyOK4 AND NOT bButtReverse4 AND (bAutomat4 OR bManual4) AND NOT bReverse4;

bDirect1:=b_1KM1_1;
bReverse1:=b_1KM1_2;
fbDirection1(bAutomat:=bAutomat1, bManual:=bManual1, bDirectOn :=bDirect1, bReverseOn:=bReverse1,
	bButtReverse:=bButtReverse1,bSwitchOnDirect=>b_1K1_1, bSwitchOnReverse=>b_1K1_2);

	
bDirect2:=b_2KM1_1;
bReverse2:=b_2KM1_2;
fbDirection2(bAutomat:=bAutomat2, bManual:=bManual2, bDirectOn :=bDirect2, bReverseOn:=bReverse2,
	bButtReverse:=bButtReverse2,bSwitchOnDirect=>b_2K1_1, bSwitchOnReverse=>b_2K1_2);
	
	
bDirect3:=b_3KM1_1;
bReverse3:=b_3KM1_2;
fbDirection3(bAutomat:=bAutomat3, bManual:=bManual3, bDirectOn :=bDirect3, bReverseOn:=bReverse3,
	bButtReverse:=bButtReverse3,bSwitchOnDirect=>b_3K1_1, bSwitchOnReverse=>b_3K1_2);
	
	
bDirect4:=b_4KM1_1;
bReverse4:=b_4KM1_2;
fbDirection4(bAutomat:=bAutomat4, bManual:=bManual4, bDirectOn :=bDirect4, bReverseOn:=bReverse4,
	bButtReverse:=bButtReverse4,bSwitchOnDirect=>b_4K1_1, bSwitchOnReverse=>b_4K1_2);
	
	
(*

IF (*bButtManu1*)bManual1 AND bButtReverse1 AND NOT b_1K1_1 THEN b_1K1_2 := TRUE;
	ELSE b_1K1_2 := FALSE;
END_IF
IF bButtManu2 AND bButtReverse2 AND NOT b_2K1_1 THEN b_2K1_2 := TRUE;
	ELSE b_2K1_2 := FALSE;
END_IF
IF bButtManu3 AND bButtReverse3 AND NOT b_3K1_1 THEN b_3K1_2 := TRUE;
	ELSE b_3K1_2 := FALSE;
END_IF
IF bButtManu4 AND bButtReverse4 AND NOT b_4K1_1 THEN b_4K1_2 := TRUE;
	ELSE b_4K1_2 := FALSE;
END_IF
*)
AlarmEventGeneral();

END_PROGRAM

// ---- POUs/FB/FB_Direction.TcPOU
FUNCTION_BLOCK FB_Direction
VAR_INPUT
	bAutomat:BOOL;
	bManual:BOOL;
	bDirectOn :BOOL;
	bReverseOn:BOOL;
	bButtReverse:BOOL;
END_VAR
VAR_OUTPUT
	bSwitchOnDirect:BOOL:=FALSE;
	bSwitchOnReverse:BOOL:=FALSE;
END_VAR
VAR
	bModeDirect:BOOL;
	bModeReverse:BOOL;
	fbPulsButt:R_TRIG;
	fbDelayOnDirect:TON;
	fbDelayOffDirect:TON;
END_VAR


fbDelayOnDirect(IN:=NOT bReverseOn, PT:=T#1S);

IF (bManual OR bAutomat) AND fbDelayOnDirect.Q(*NOT bReverseOn*) THEN
	bSwitchOnDirect:=TRUE;
END_IF
IF NOT (bManual OR bAutomat) THEN 
	bSwitchOnDirect:=FALSE;
END_IF

 fbDelayOffDirect(IN:=NOT bDirectOn, PT:=T#1S);   

fbPulsButt(CLK:=bButtReverse  );
IF fbPulsButt.Q AND bManual AND NOT bModeReverse  THEN
bModeReverse:=TRUE;
END_IF
IF bModeReverse THEN
	bSwitchOnDirect:=FALSE;
	IF NOT bSwitchOnDirect AND (*NOT bDirectOn*)fbDelayOffDirect.Q THEN
		bSwitchOnReverse:=TRUE;
	END_IF
END_IF

IF fbPulsButt.Q AND bReverseOn  THEN
	bSwitchOnReverse:=FALSE;
	bModeReverse :=FALSE;
END_IF

END_FUNCTION_BLOCK

// ---- POUs/Alarms/AlarmEventGeneral.TcPOU
PROGRAM AlarmEventGeneral
VAR
	fbEventlogger					:FB_TcEventLogger;
	fbAlarm							:FB_TcAlarm;
	fbAlarm1						:FB_TcAlarm;
	fbMessage						:FB_TcMessage;
	bMessage						:BOOL;
	bIsInitalized					:BOOL;
	bClearAlarm						:BOOL;
	bConfirmAlarm					:BOOL;

//Нет готовности БП
	fbNotReadyPower24v				:FB_TcAlarm;
//УЗИП	
	fbAlarm1QF						:FB_TcAlarm;
	fbAlarm2QF						:FB_TcAlarm;

	fbAlarmSF3						:FB_TcAlarm;
	fbAlarmSF3_						:FB_TcAlarm;
//Аварии ввода	
	fbAlarmK2						:FB_TcAlarm;
	fbAlarmK2_						:FB_TcAlarm;
//Реле безопасности		
	fbAlarm1AS1						:FB_TcAlarm;
	fbAlarm2AS1						:FB_TcAlarm;
	fbAlarm3AS1						:FB_TcAlarm;
	fbAlarm4AS1						:FB_TcAlarm;
//Питание приводов	
	fbAlarm1QF1						:FB_TcAlarm;
	fbAlarm2QF1						:FB_TcAlarm;
	fbAlarm3QF1						:FB_TcAlarm;
	fbAlarm4QF1						:FB_TcAlarm;
//Превышение тока или напряжения	
	fbAlarm1P_I						:FB_TcAlarm;
	fbAlarm1P_U						:FB_TcAlarm;
//-----------------------------------------------------------------------------------------//	
 	fbButtAlarmResetGeneral_RTRIG	:R_TRIG;
 	fbbButtAlarmReset1_RTRIG		:R_TRIG;

//Нет готовности БП
	fbExecNotReadyPower24v			:FB_AlarmEvent;
//УЗИП	
	fbExecAlarm1QF					:FB_AlarmEvent;
	fbExecAlarm2QF					:FB_AlarmEvent;
	
	fbExecAlarmSF3					:FB_AlarmEvent;
	fbExecAlarmSF3_					:FB_AlarmEvent;
//Аварии ввода	
	fbExecAlarmK2					:FB_AlarmEvent;
	fbExecAlarmK2_					:FB_AlarmEvent;
//Реле безопасности	
	fbExecAlarm1AS1					:FB_AlarmEvent;
	fbExecAlarm2AS1					:FB_AlarmEvent;
	fbExecAlarm3AS1					:FB_AlarmEvent;
	fbExecAlarm4AS1					:FB_AlarmEvent;
//Питание приводов	
	fbExecAlarm1QF1					:FB_AlarmEvent;
	fbExecAlarm2QF1					:FB_AlarmEvent;
	fbExecAlarm3QF1					:FB_AlarmEvent;
	fbExecAlarm4QF1					:FB_AlarmEvent;
//Превышение тока или напряжения	
	fbExecAlarm1P_I					:FB_AlarmEvent;
	fbExecAlarm1P_U					:FB_AlarmEvent;
END_VAR

Initialization();

fbButtAlarmResetGeneral_RTRIG(CLK := bButtAlarmResetGeneral);

fbExecNotReadyPower24v(bAlarmEvent :=bNotReadyPower24v, bButtAlarmReset:=fbButtAlarmResetGeneral_RTRIG.Q, fbAlarm:=fbNotReadyPower24v);

fbExecAlarm1QF(bAlarmEvent :=bAlarm1QF, bButtAlarmReset:=fbButtAlarmResetGeneral_RTRIG.Q, fbAlarm:=fbAlarm1QF);
fbExecAlarm2QF(bAlarmEvent :=bAlarm2QF, bButtAlarmReset:=fbButtAlarmResetGeneral_RTRIG.Q, fbAlarm:=fbAlarm2QF);

fbExecAlarmSF3(bAlarmEvent :=bAlarmSF3, bButtAlarmReset:=fbButtAlarmResetGeneral_RTRIG.Q, fbAlarm:=fbAlarmSF3);
fbExecAlarmSF3_(bAlarmEvent :=bAlarmSF3_, bButtAlarmReset:=fbButtAlarmResetGeneral_RTRIG.Q, fbAlarm:=fbAlarmSF3_);

fbExecAlarmK2(bAlarmEvent :=bAlarmK2, bButtAlarmReset:=fbButtAlarmResetGeneral_RTRIG.Q, fbAlarm:=fbAlarmK2);
fbExecAlarmK2_(bAlarmEvent :=bAlarmK2_, bButtAlarmReset:=fbButtAlarmResetGeneral_RTRIG.Q, fbAlarm:=fbAlarmK2_);

fbExecAlarm1AS1(bAlarmEvent :=bAlarm1AS1, bButtAlarmReset:=fbButtAlarmResetGeneral_RTRIG.Q, fbAlarm:=fbAlarm1AS1);
fbExecAlarm2AS1(bAlarmEvent :=bAlarm2AS1, bButtAlarmReset:=fbButtAlarmResetGeneral_RTRIG.Q, fbAlarm:=fbAlarm2AS1);
fbExecAlarm3AS1(bAlarmEvent :=bAlarm3AS1, bButtAlarmReset:=fbButtAlarmResetGeneral_RTRIG.Q, fbAlarm:=fbAlarm3AS1);
fbExecAlarm4AS1(bAlarmEvent :=bAlarm4AS1, bButtAlarmReset:=fbButtAlarmResetGeneral_RTRIG.Q, fbAlarm:=fbAlarm4AS1);

fbExecAlarm1QF1(bAlarmEvent :=bAlarm1QF1, bButtAlarmReset:=fbButtAlarmResetGeneral_RTRIG.Q, fbAlarm:=fbAlarm1QF1);
fbExecAlarm2QF1(bAlarmEvent :=bAlarm2QF1, bButtAlarmReset:=fbButtAlarmResetGeneral_RTRIG.Q, fbAlarm:=fbAlarm2QF1);
fbExecAlarm3QF1(bAlarmEvent :=bAlarm3QF1, bButtAlarmReset:=fbButtAlarmResetGeneral_RTRIG.Q, fbAlarm:=fbAlarm3QF1);
fbExecAlarm4QF1(bAlarmEvent :=bAlarm4QF1, bButtAlarmReset:=fbButtAlarmResetGeneral_RTRIG.Q, fbAlarm:=fbAlarm4QF1);

fbExecAlarm1P_I(bAlarmEvent :=bAlarm1P_I, bButtAlarmReset:=fbButtAlarmResetGeneral_RTRIG.Q, fbAlarm:=fbAlarm1P_I);
fbExecAlarm1P_U(bAlarmEvent :=bAlarm1P_U, bButtAlarmReset:=fbButtAlarmResetGeneral_RTRIG.Q, fbAlarm:=fbAlarm1P_U);

ACTION Initialization:
IF NOT bIsInitalized THEN
	bIsInitalized := TRUE;

	fbNotReadyPower24v.CreateEx(TC_Events.AlarmGeneral.NotReadyPower24v, TRUE, 0);
	
	fbAlarm1QF.CreateEx(TC_Events.AlarmGeneral.Alarm1QF, TRUE, 0);
	fbAlarm2QF.CreateEx(TC_Events.AlarmGeneral.Alarm2QF, TRUE, 0);
	
	fbAlarmSF3.CreateEx(TC_Events.AlarmGeneral.AlarmSF3, TRUE, 0);
	fbAlarmSF3_.CreateEx(TC_Events.AlarmGeneral.AlarmSF3_, TRUE, 0);
	
	fbAlarmK2.CreateEx(TC_Events.AlarmGeneral.AlarmK2, TRUE, 0);
	fbAlarmK2_.CreateEx(TC_Events.AlarmGeneral.AlarmK2_, TRUE, 0);
	
	fbAlarm1AS1.CreateEx(TC_Events.AlarmGeneral.Alarm1AS1, TRUE, 0);
	fbAlarm2AS1.CreateEx(TC_Events.AlarmGeneral.Alarm2AS1, TRUE, 0);
	fbAlarm3AS1.CreateEx(TC_Events.AlarmGeneral.Alarm3AS1, TRUE, 0);
	fbAlarm4AS1.CreateEx(TC_Events.AlarmGeneral.Alarm4AS1, TRUE, 0);
	
	fbAlarm1QF1.CreateEx(TC_Events.AlarmGeneral.Alarm1QF1, TRUE, 0);
	fbAlarm2QF1.CreateEx(TC_Events.AlarmGeneral.Alarm2QF1, TRUE, 0);
	fbAlarm3QF1.CreateEx(TC_Events.AlarmGeneral.Alarm3QF1, TRUE, 0);
	fbAlarm4QF1.CreateEx(TC_Events.AlarmGeneral.Alarm4QF1, TRUE, 0);
	
	fbAlarm1P_I	.CreateEx(TC_Events.AlarmGeneral.Alarm1P_I, TRUE, 0);
	fbAlarm1P_U	.CreateEx(TC_Events.AlarmGeneral.Alarm1P_U, TRUE, 0);
	
END_IF
END_ACTION

END_PROGRAM

// ---- POUs/ExchangeWMS/Exchange_WMS.TcPOU
PROGRAM Exchange_WMS

VAR_INPUT
	
END_VAR
VAR
	
fbFileOpen:FB_FileOpen;
iStep:INT;
bFileOpen:BOOL;
fbPulsWriteMessage:R_TRIG;
bError1:BOOL;
nErrId1:UDINT;
hFile  : UINT;    
fbFileWrite: FB_FileWrite;
bError2:BOOL;
nErrId2:UDINT;

fbFileClose:FB_FileClose;
bError3:BOOL;
nErrId3:UDINT;

bSendToWMS:BOOL;
fbUpload_ToServer:FB_Upload_ToServer;


fbTime : FB_LocalSystemTime;
	System_Time: DT;
	bEnableTime: BOOL := TRUE;
tNow : TIME;

sSystemTimeYear:STRING;
sSystemTimeMonth:STRING;

bSendToWMS_OK: BOOL ;
fbPulsSend_OK:R_TRIG;
sSystemTime1:STRING;
sPathName:STRING;
sSrcFile:STRING;
sDesFile:STRING;

fbTail: FB_Tail;
bMessageReady:BOOL;
 bReset:BOOL;
 bShiftBuff:BOOL;
 sMessageOut: T_MaxString;
 sMessageOutStore: T_MaxString;
 bNew:BOOL;
 bTest:BOOL;
END_VAR




fbTime  (bEnable :=bEnableTime , dwCycle :=1);
bEnableTime := FALSE;

System_Time := SYSTEMTIME_TO_DT (fbTime.systemTime);
sSystemTime := DT_TO_STRING (System_Time);
sSystemTime := MID (sSystemTime, 19, 4);
sSystemTime1 := sSystemTime;
sSystemTimeYear :=LEFT(sSystemTime,4);
sSystemTimeMonth:=MID(sSystemTime,2,6);
sSystemTime := MID (sSystemTime, 11, 9);
sSystemTime:= REPLACE(sSystemTime,CONCAT('.',sSystemTimeMonth),1,3);
sSystemTime:= INSERT(sSystemTime,CONCAT(CONCAT('.',sSystemTimeYear),' '),5);






fbTail(sMessage1:=sMessageOut1,
	sMessage2:=sMessageOut2,
	sMessage3:=sMessageOut3,
	sMessage4:=sMessageOut4,
    bReset:=bReset,	bMessageReady1:=bMessageReady1,
	bMessageReady2:=bMessageReady2,
	bMessageReady3:=bMessageReady3,
	bMessageReady4:=bMessageReady4,
	bShiftBuff:=bShiftBuff,sMessageOut:=sMessageOut,bNew:=bNew);

	
(*	
IF bNew	THEN
	IF sMessageOut<>'' THEN
		bMessageReady:=TRUE;
	END_IF
	bNew:=FALSE;
END_IF
*)	
bMessageReady:=(*bNew	*)sMessageOut<>sMessageOutStore AND sMessageOut<>'' AND NOT  bShiftBuff;

fbPulsWriteMessage(CLK:=bMessageReady);
IF fbPulsWriteMessage.Q THEN
	
sMessageOutStore:=sMessageOut;
//bMessageReady:=FALSE;

sSystemTime1:=REPLACE(sSystemTime1,'_',1, 11);
sSystemTime1:=REPLACE(sSystemTime1,'-',1, 14);
sSystemTime1:=REPLACE(sSystemTime1,'-',1, 17);
sPathName:= INSERT ('C:\FTPclient\out\WMS_.in',sSystemTime1,21 );



bTest:=TRUE;

	iStep:=1;
END_IF
CASE iStep OF

0: ;

1:
bSendToWMS:=FALSE;
fbFileOpen(bExecute:= FALSE,);
fbFileOpen( sPathName :=  sPathName(*'C:\FTPclient\out\WMS_Line1.in'*),  nMode:= FOPEN_MODEWRITE,                                
            bExecute:= TRUE,tTimeout:=T#3S );
iStep:=2;

2:
  fbFileOpen( bExecute := FALSE );
                IF NOT fbFileOpen.bBusy THEN
                        IF fbFileOpen.bError THEN
                                nErrId1 := fbFileOpen.nErrId;
                                bError1 := TRUE;
                                iStep := 50;
                        ELSE
                                hFile := fbFileOpen.hFile;
                                iStep := 3;
                        END_IF
                END_IF
				
3:
fbFileWrite( bExecute := FALSE );
                fbFileWrite(  hFile:=hFile,
                        pWriteBuff:= ADR(sMessageOut), cbWriteLen:= LEN(sMessageOut),
                        bExecute:=TRUE, tTimeout:=T#3S  );
                iStep := 4;				
				
4:
fbFileWrite( bExecute := FALSE );
                 IF NOT fbFileWrite.bBusy THEN
                        IF fbFileWrite.bError THEN
                                nErrId2 := fbFileWrite.nErrId;
                                bError2 := TRUE;
                                iStep := 50;
								
                        ELSE
                               // IF fbFileRead.bEOF THEN (* Check if the EOF flag ist set *)
                                 iStep := 5;(* Cleanup: close the destination and source files *)
                       // sMessageOut:='';
                         
                        END_IF
                END_IF
5:
  fbFileClose( bExecute := FALSE );
                fbFileClose(  hFile:=hFile, bExecute:=TRUE, tTimeout:=T#3S );
                iStep := 6;
				
6:
                fbFileClose( bExecute := FALSE );
                IF NOT fbFileClose.bBusy THEN
                        IF fbFileClose.bError THEN
                                nErrId3 := fbFileClose.nErrId;
                                bError3 := TRUE;
                        END_IF
                        iStep := 7;
                        hFile := 0;
                END_IF		
		
7:
       bSendToWMS:=TRUE;
		 iStep := 0;
         bShiftBuff:=TRUE;		
50:;				
END_CASE
sSrcFile:=sPathName;

sDesFile:=CONCAT('\in\', RIGHT(sSrcFile,26));

fbUpload_ToServer(bStartstop:=bSendToWMS,sHost:='10.45.19.159'(*'10.45.19.5'*),sDesFile:=sDesFile ,sSrcFile:=sSrcFile, bSendToWMS_OK=>bSendToWMS_OK );

END_PROGRAM

// ---- POUs/ExchangeWMS/FB_Upload_ToServer.TcPOU
FUNCTION_BLOCK FB_Upload_ToServer
VAR_INPUT
	bStartstop 			: BOOL;
	sHost :STRING;
	sUsername:STRING:=(*'FTPclient';*)'CX-4F6D58';
	sPassword:STRING:= 'Fabslog8721';
	sSrcFile:STRING:= '\FTPclient\out\WMS_Line1.in';
	sDesFile:STRING:= '\in\WMS_Line1.in';
END_VAR
VAR_OUTPUT
	err1 				: BOOL;
	errid1 				: UDINT;
	err2				: BOOL;
	errid2 				: UDINT;
	err3				: BOOL;
	errid3				: UDINT;
	err4				: BOOL;
	errid4				: UDINT;
	bSendToWMS_OK       : BOOL;
END_VAR
VAR
	RisingEdge 			: R_TRIG;
	
	state				: BYTE;
	fbFTP_Open1 		: FB_FTP_OpenEX;
	fbFTPFileUpload1: FB_FTP_FileUpload;
	fbFTP_Close1 		: FB_FTP_Close;
	busy1 				: BOOL;
busy2				: BOOL;
busy3 				: BOOL;
busy4 				: BOOL;
	handle 				: T_HFTP;
	progress 			: UDINT;
fbFTP_FileExist:FB_FTP_FileExist;
bFileExist:BOOL;
END_VAR

RisingEdge(CLK:= bStartstop);
IF RisingEdge.Q THEN
	state := 1;
END_IF

CASE state OF
	0:
		;

	1:
	bSendToWMS_OK :=FALSE;
		fbFTP_Open1(
			sNetID:= ,
			sHost:= sHost,
			nPort:= 21,
			sUsername:= sUsername,
	        sPassword:= sPassword,
			bExecute:= TRUE,
			tTimeout:= T#15S,
			 eMode    := 1,
			bBusy=> busy1,
			bError=> err1,
			nErrId=> errid1,
			hFTP=> handle);

		IF NOT busy1 AND NOT err1 THEN
			fbFTP_Open1(bExecute:= FALSE);
			state := 3;
		
				
		END_IF
		
2: 
fbFTP_FileExist(
 hFTP:=handle,
sFile:=sDesFile,
bExecute:= TRUE,
	tTimeout:= T#15s,
	bBusy=> busy4,
	bError=> err4,
	nErrId=> errid4,
	bExist=> bFileExist);
		
		IF NOT busy4 AND NOT err4 THEN
			fbFTP_FileExist(bExecute:= FALSE);
			IF NOT bFileExist THEN
			state := 3;
			ELSE
				state := 1;
			END_IF
		END_IF

		
		
		
		
	3:
		fbFTPFileUpload1(
	sNetID:='' ,
     hFTP:=handle,
	sSrcFile:= sSrcFile,
	sDesFile:=sDesFile,
	bExecute:= TRUE,
	tTimeout:= T#15s,
	bBusy=> busy2,
	bError=> err2,
	nErrId=> errid2,
	nProgress=> progress);

		IF NOT busy2 AND NOT err2 THEN
			fbFTPFileUpload1(bExecute:= FALSE);
			state := 4;
		END_IF

	4:
		fbFTP_Close1(
			sNetID:= ,
			hFTP:= handle,
			bExecute:= TRUE,
			tTimeout:= T#15s,
			bBusy => busy3,
			bError => err3,
			nErrId => errid3);

		IF NOT busy3 AND NOT err3 THEN
			fbFTP_Close1(bExecute:= FALSE);
			state := 0;
			bSendToWMS_OK :=TRUE;
		END_IF

END_CASE

END_FUNCTION_BLOCK

// ---- POUs/ExchangeWMS/FB_Tail.TcPOU
FUNCTION_BLOCK FB_Tail
VAR_INPUT
	sMessage1 :T_MaxString;
	sMessage2 :T_MaxString;
	sMessage3 :T_MaxString;
	sMessage4 :T_MaxString;
    bReset:BOOL;
END_VAR
VAR_OUTPUT
	
	
END_VAR
VAR
	fbBuffer:FB_TransBuffer;
	aTransBuff : ARRAY[1..10] OF T_MaxString;
	
	bReady:BOOL;
	bEmpty:BOOL;
END_VAR
VAR_IN_OUT
	bMessageReady1:BOOL;
	bMessageReady2:BOOL;
	bMessageReady3:BOOL;
	bMessageReady4:BOOL;
	bShiftBuff:BOOL;
	sMessageOut:T_MaxString;
	bNew:BOOL;
END_VAR


IF bMessageReady1 AND NOT fbBuffer.bBusy  THEN
	fbBuffer(sTrans:=sMessage1,bWriteInBuff:=bMessageReady1,aTransBuff:=aTransBuff,bShiftBuff:=bShiftBuff,bNew:=bNew);
END_IF
IF bMessageReady2 AND NOT fbBuffer.bBusy  THEN
	fbBuffer(sTrans:=sMessage2,bWriteInBuff:=bMessageReady2,aTransBuff:=aTransBuff,bShiftBuff:=bShiftBuff,bNew:=bNew);
END_IF
IF bMessageReady3 AND NOT fbBuffer.bBusy  THEN
	fbBuffer(sTrans:=sMessage3,bWriteInBuff:=bMessageReady3,aTransBuff:=aTransBuff,bShiftBuff:=bShiftBuff,bNew:=bNew);
END_IF
IF bMessageReady4 AND NOT fbBuffer.bBusy  THEN
	fbBuffer(sTrans:=sMessage4,bWriteInBuff:=bMessageReady4,aTransBuff:=aTransBuff,bShiftBuff:=bShiftBuff,bNew:=bNew);
END_IF





(*
IF bMessageReady1 AND NOT fbBuffer.bBusy  THEN
	fbBuffer(sTrans:=sMessage1,bWriteInBuff:=bMessageReady1,aTransBuff:=aTransBuff,bShiftBuff:=bShiftBuff);
   IF	NOT fbBuffer.bBusy THEN
	   bReady:=TRUE;
   END_IF
   
   
   
ELSIF bMessageReady2 AND NOT fbBuffer.bBusy THEN
	fbBuffer(sTrans:=sMessage2,bWriteInBuff:=bMessageReady2,aTransBuff:=aTransBuff,bShiftBuff:=bShiftBuff);
	  IF	NOT fbBuffer.bBusy THEN
	   bReady:=TRUE;
   END_IF 
ELSIF bMessageReady3 THEN
	fbBuffer(sTrans:=sMessage3,bWriteInBuff:=bMessageReady3,aTransBuff:=aTransBuff,bShiftBuff:=bShiftBuff);	
ELSIF bMessageReady4 THEN
	fbBuffer(sTrans:=sMessage4,bWriteInBuff:=bMessageReady4,aTransBuff:=aTransBuff,bShiftBuff:=bShiftBuff);	
	*)
	
(*IF 	NOT fbBuffer.bBusy  THEN
	fbBuffer(sTrans:=sMessage1,bWriteInBuff:=bMessageReady1,aTransBuff:=aTransBuff,bShiftBuff:=bEmpty);
	fbBuffer(sTrans:=sMessage2,bWriteInBuff:=bMessageReady2,aTransBuff:=aTransBuff,bShiftBuff:=bEmpty);
    fbBuffer(sTrans:=sMessage3,bWriteInBuff:=bMessageReady3,aTransBuff:=aTransBuff,bShiftBuff:=bEmpty);	
    fbBuffer(sTrans:=sMessage4,bWriteInBuff:=bMessageReady4,aTransBuff:=aTransBuff,bShiftBuff:=bEmpty);	
    fbBuffer(bWriteInBuff:=bEmpty,aTransBuff:=aTransBuff,bShiftBuff:=bShiftBuff);
END_IF*)
	
   fbBuffer(bWriteInBuff:=bEmpty,aTransBuff:=aTransBuff,bShiftBuff:=bShiftBuff,bReset:=bReset,bNew:=bNew);
   
	sMessageOut:=fbBuffer.sTransBuffOut;

END_FUNCTION_BLOCK

// ---- POUs/ExchangeWMS/FB_TransBuffer.TcPOU
FUNCTION_BLOCK FB_TransBuffer
VAR_INPUT
	
    sTrans: T_MaxString;
	
	bReset : BOOL;
END_VAR
VAR_OUTPUT
	sTransBuffOut :T_MaxString;
    bBusy: BOOL;
END_VAR
VAR
	i: INT;
	j: INT;
	k: INT;
	bGoodWrite: BOOL;
	bRiseReset: BOOL;
	
END_VAR
VAR_IN_OUT
	bWriteInBuff : BOOL;
	bShiftBuff : BOOL;
	aTransBuff : ARRAY[1..10] OF T_MaxString;
	bNew:BOOL;
END_VAR


IF bWriteInBuff THEN
bBusy:=TRUE;
FOR j:=1 TO 10 DO
IF aTransBuff[j] = '' THEN
aTransBuff[j] :=  sTrans;
IF J=1 THEN
	bNew:=TRUE;
END_IF

EXIT;
END_IF
END_FOR
bWriteInBuff :=FALSE;
bBusy:=FALSE;
END_IF




IF bShiftBuff THEN
bBusy:=TRUE;
FOR i:=1 TO 9 DO aTransBuff[i] :=aTransBuff[i+1];
END_FOR

aTransBuff[10]:='';
bShiftBuff := FALSE;
bBusy:=FALSE;
bNew:=TRUE;
END_IF

sTransBuffOut := aTransBuff[1];

IF bReset  THEN
FOR k :=1 TO 10 DO
aTransBuff[k] :='';
END_FOR

END_IF
bReset := FALSE;

END_FUNCTION_BLOCK

// ---- POUs/ConvLine1.TcPOU
PROGRAM ConvLine1
VAR_INPUT
	bAutomat				:BOOL;
	bManual					:BOOL;
	bStop					:BOOL;
	bReset					:BOOL := FALSE;
	bDirect					:BOOL;
	bReverse				:BOOL;
	bBuffering				:BOOL;
END_VAR
VAR
	fbS1			:FB_ConvPlace;
	fbS2			:FB_ConvPlaceDouble;
	fbS3			:FB_ConvPlaceDouble;
	fbS4			:FB_ConvPlaceDouble;
	fbS5			:FB_ConvPlace;
	fbS6			:FB_ConvPlace;
	bMove1					:BOOL;
	bMove2					:BOOL;
	bDriveMoveS1			:BOOL;
	bDriveMoveS2			:BOOL;
	bEnableMoveToS1			:BOOL :=TRUE;
	bEnableMoveToS2			:BOOL;
	bEnableMoveToS3			:BOOL;
	bEnableMoveToS4			:BOOL;
	bEnableMoveToS5			:BOOL;
	bEnableMoveToS6			:BOOL;
	bEnableRead				:BOOL;
	bEnableWeight			:BOOL;
	fbLoadScan				:FB_LoadScan;
	fbLoadWeight			:FB_LoadWeight;
	bEnableReadyID			:BOOL;
	bEnableReadyData		:BOOL;
	ConvStatusPrev 			:BYTE;
	bSensFreePrevS1 		:BOOL;
	bSensFreePrevS5 		:BOOL;
	bSensFreePrevS6 		:BOOL;

	bCountNoRead_ID1		:WORD;		//Кол-во несчитываний RFID
	bSetVal_ID1				:WORD :=10;	//Заданное значение счетчика (максимально допустимое для несчитываний)
	bResetCTU_ID1			:BOOL;		//Сброс счетчика несчитываний
	
	bCountNoRead_Weight1	:WORD;		//Кол-во несчитываний RFID
	bSetVal_Weight1			:WORD :=10;	//Заданное значение счетчика (максимально допустимое для несчитываний)
	bResetCTU_Weight1		:BOOL;		//Сброс счетчика несчитываний
	
	fbLoadDataToWMS: FB_LoadDataToWMS;
	
	bEnableMove3_2:BOOL;
	bEnableMove3_3:BOOL;
	bEnableMove3_4:BOOL;
	
	fbDelayEnableMove3_2:TON;
	fbDelayEnableMove3_3:TON;
	fbDelayEnableMove3_4:TON;
	
	
	fbFallMove1:F_TRIG;
	fbFallMove2:F_TRIG;
	bLineFree:BOOL;
	fbFreeS6:R_TRIG;
END_VAR
VAR PERSISTENT
	iCounterPallets:INT;
END_VAR




fbS1 ( bAutomat:=bAutomat, bManual:=bManual,bStop:=bStop,bReset:=bReset,tBusy:=T#6S, bFirstPlace:=TRUE,
       	bDriveMove:=fbS2.bDrivePrev, bSens1:=bSens1s01D2, bSens2:=bSens1s01D1, bDirect:=bDirect	,bReverse:=bReverse,
       	bSensFork:= bSens1s01D3, bButtConv:= bButt1s01,bButtConvRev:=bButt1s01Rev,
	  	bMove:=bMove1,ConvStatusPrev:=ConvStatusPrev, bEnableMove := bEnableMoveToS1, bSensFreePrev := bSensFreePrevS1);
	  
		bSensFreePrevS1 := fbS1.ConvStatus = 0;
	  	bEnableMoveToS2:= NOT bMove1s02_2_s03_1 AND NOT bMove1s02_s03;
	  
		bLineFree:= fbS3.ConvStatus1=0 AND fbS3.ConvStatus2=0 AND 
      fbS4.ConvStatus1=0 AND fbS4.ConvStatus2=0 AND NOT (bMove1s02_2_s03_1 OR bMove1s02_s03 OR bMove1s03_1_s03_2
      OR bMove1s03_2_s04_1 OR bMove1s03_s04 OR bMove1s04_1_s04_2  OR bMove1s05_s06 OR bMove1s04_2_s05);	 
	  
 IF bLineFree AND fbS6.ConvStatus=0 AND fbS5.ConvStatus=0 THEN
	 iCounterPallets:=0;
 END_IF
	  
		fbFallMove1(CLK:=bMove1s02_2_s03_1);
IF fbFallMove1.Q THEN	
iCounterPallets:=iCounterPallets +1;
END_IF	
	   fbFallMove2(CLK:=bMove1s02_s03);
IF 	fbFallMove2.Q   THEN
	iCounterPallets:=iCounterPallets +2;
END_IF



		fbFreeS6(CLK:=fbS6.ConvStatus=0);
IF fbFreeS6.Q AND iCounterPallets>0 THEN
iCounterPallets:=iCounterPallets -1;	
END_IF

		
		bEnableMove3_2 := (*(fbS6.ConvStatus=0 OR fbS5.ConvStatus=0) AND bLineFree OR *)iCounterPallets<2;
	//  fbDelayEnableMove3_2(IN:=bEnableMove3_2, PT:=T#0.3S);
		
	  
	
	
	  
